  PROC DrawPart24()
    MoveL Offs(pOrigin,312.39,170.23,0.00),v60,z0,tPen\WObj:=wPaper;
    MoveL Offs(pOrigin,314.80,167.82,0.00),v40,z0,tPen\WObj:=wPaper;
    MoveL Offs(pOrigin,313.96,168.12,0.00),v40,z0,tPen\WObj:=wPaper;
    MoveL Offs(pOrigin,312.90,168.12,0.00),v40,fine,tPen\WObj:=wPaper;
    MoveL Offs(pOrigin,312.90,168.12,6.00),v60,z5,tPen\WObj:=wPaper;
    MoveL Offs(pOrigin,312.51,169.44,6.00),vTravel,z5,tPen\WObj:=wPaper;
    MoveL Offs(pOrigin,312.51,169.44,0.00),v60,z0,tPen\WObj:=wPaper;
    MoveL Offs(pOrigin,315.82,172.74,0.00),v40,z0,tPen\WObj:=wPaper;
    MoveL Offs(pOrigin,316.28,172.31,0.00),v40,z0,tPen\WObj:=wPaper;
    MoveL Offs(pOrigin,313.88,174.72,0.00),v40,z0,tPen\WObj:=wPaper;
    MoveL Offs(pOrigin,314.02,173.94,0.00),v40,z0,tPen\WObj:=wPaper;
    MoveL Offs(pOrigin,317.48,177.39,0.00),v40,z0,tPen\WObj:=wPaper;
    MoveL Offs(pOrigin,317.15,177.62,0.00),v40,z0,tPen\WObj:=wPaper;
    MoveL Offs(pOrigin,316.09,177.62,0.00),v40,z0,tPen\WObj:=wPaper;
    MoveL Offs(pOrigin,315.66,176.57,0.00),v40,z0,tPen\WObj:=wPaper;
    MoveL Offs(pOrigin,316.73,176.57,0.00),v40,z0,tPen\WObj:=wPaper;
    MoveL Offs(pOrigin,317.92,176.65,0.00),v40,z0,tPen\WObj:=wPaper;
    MoveL Offs(pOrigin,315.36,179.21,0.00),v40,z0,tPen\WObj:=wPaper;
    MoveL Offs(pOrigin,315.81,180.25,0.00),v40,z0,tPen\WObj:=wPaper;
    MoveL Offs(pOrigin,320.62,175.44,0.00),v40,z0,tPen\WObj:=wPaper;
    MoveL Offs(pOrigin,320.17,174.40,0.00),v40,z0,tPen\WObj:=wPaper;
    MoveL Offs(pOrigin,318.82,175.75,0.00),v40,fine,tPen\WObj:=wPaper;
    MoveL Offs(pOrigin,318.82,175.75,6.00),v60,z5,tPen\WObj:=wPaper;
    MoveL Offs(pOrigin,318.67,174.40,6.00),vTravel,z5,tPen\WObj:=wPaper;
    MoveL Offs(pOrigin,318.67,174.40,0.00),v60,z0,tPen\WObj:=wPaper;
    MoveL Offs(pOrigin,319.57,173.50,0.00),v40,fine,tPen\WObj:=wPaper;
    MoveL Offs(pOrigin,319.57,173.50,6.00),v60,z5,tPen\WObj:=wPaper;
    MoveL Offs(pOrigin,317.02,174.56,6.00),vTravel,z5,tPen\WObj:=wPaper;
    MoveL Offs(pOrigin,317.02,174.56,0.00),v60,z0,tPen\WObj:=wPaper;
    MoveL Offs(pOrigin,314.62,176.96,0.00),v40,z0,tPen\WObj:=wPaper;
    MoveL Offs(pOrigin,314.63,176.03,0.00),v40,z0,tPen\WObj:=wPaper;
    MoveL Offs(pOrigin,318.08,179.49,0.00),v40,z0,tPen\WObj:=wPaper;
    MoveL Offs(pOrigin,317.79,179.74,0.00),v40,z0,tPen\WObj:=wPaper;
    MoveL Offs(pOrigin,316.73,179.74,0.00),v40,z0,tPen\WObj:=wPaper;
    MoveL Offs(pOrigin,316.14,180.53,0.00),v40,z0,tPen\WObj:=wPaper;
    MoveL Offs(pOrigin,318.54,182.94,0.00),v40,z0,tPen\WObj:=wPaper;
    MoveL Offs(pOrigin,317.58,182.90,0.00),v40,z0,tPen\WObj:=wPaper;
    MoveL Offs(pOrigin,315.02,182.90,0.00),v40,z0,tPen\WObj:=wPaper;
    MoveL Offs(pOrigin,315.10,182.48,0.00),v40,z0,tPen\WObj:=wPaper;
    MoveL Offs(pOrigin,316.75,184.13,0.00),v40,fine,tPen\WObj:=wPaper;
    MoveL Offs(pOrigin,316.75,184.13,6.00),v60,z5,tPen\WObj:=wPaper;
    MoveL Offs(pOrigin,314.60,183.96,6.00),vTravel,z5,tPen\WObj:=wPaper;
    MoveL Offs(pOrigin,314.60,183.96,0.00),v60,z0,tPen\WObj:=wPaper;
    MoveL Offs(pOrigin,311.84,183.96,0.00),v40,z0,tPen\WObj:=wPaper;
    MoveL Offs(pOrigin,311.96,183.82,0.00),v40,z0,tPen\WObj:=wPaper;
    MoveL Offs(pOrigin,313.31,185.17,0.00),v40,z0,tPen\WObj:=wPaper;
    MoveL Offs(pOrigin,313.39,185.65,0.00),v40,z0,tPen\WObj:=wPaper;
    MoveL Offs(pOrigin,321.21,177.84,0.00),v40,fine,tPen\WObj:=wPaper;
    MoveL Offs(pOrigin,321.21,177.84,6.00),v60,z5,tPen\WObj:=wPaper;
    MoveL Offs(pOrigin,320.91,176.64,6.00),vTravel,z5,tPen\WObj:=wPaper;
    MoveL Offs(pOrigin,320.91,176.64,0.00),v60,z0,tPen\WObj:=wPaper;
    MoveL Offs(pOrigin,311.00,186.56,0.00),v40,z0,tPen\WObj:=wPaper;
    MoveL Offs(pOrigin,311.06,185.91,0.00),v40,z0,tPen\WObj:=wPaper;
    MoveL Offs(pOrigin,309.56,184.41,0.00),v40,z0,tPen\WObj:=wPaper;
    MoveL Offs(pOrigin,309.51,183.57,0.00),v40,z0,tPen\WObj:=wPaper;
    MoveL Offs(pOrigin,302.74,190.33,0.00),v40,z0,tPen\WObj:=wPaper;
    MoveL Offs(pOrigin,303.64,190.93,0.00),v40,z0,tPen\WObj:=wPaper;
    MoveL Offs(pOrigin,311.30,183.26,0.00),v40,z0,tPen\WObj:=wPaper;
    MoveL Offs(pOrigin,310.61,183.96,0.00),v40,z0,tPen\WObj:=wPaper;
    MoveL Offs(pOrigin,312.26,185.61,0.00),v40,z0,tPen\WObj:=wPaper;
    MoveL Offs(pOrigin,311.41,185.02,0.00),v40,z0,tPen\WObj:=wPaper;
    MoveL Offs(pOrigin,308.86,185.02,0.00),v40,z0,tPen\WObj:=wPaper;
    MoveL Offs(pOrigin,308.51,184.85,0.00),v40,z0,tPen\WObj:=wPaper;
    MoveL Offs(pOrigin,310.02,186.36,0.00),v40,fine,tPen\WObj:=wPaper;
    MoveL Offs(pOrigin,310.02,186.36,6.00),v60,z5,tPen\WObj:=wPaper;
    MoveL Offs(pOrigin,308.23,186.07,6.00),vTravel,z5,tPen\WObj:=wPaper;
    MoveL Offs(pOrigin,308.23,186.07,0.00),v60,z0,tPen\WObj:=wPaper;
    MoveL Offs(pOrigin,305.68,186.07,0.00),v40,z0,tPen\WObj:=wPaper;
    MoveL Offs(pOrigin,305.07,185.89,0.00),v40,z0,tPen\WObj:=wPaper;
    MoveL Offs(pOrigin,306.57,187.39,0.00),v40,z0,tPen\WObj:=wPaper;
    MoveL Offs(pOrigin,305.68,187.13,0.00),v40,z0,tPen\WObj:=wPaper;
    MoveL Offs(pOrigin,302.91,187.13,0.00),v40,z0,tPen\WObj:=wPaper;
    MoveL Offs(pOrigin,302.98,186.78,0.00),v40,z0,tPen\WObj:=wPaper;
    MoveL Offs(pOrigin,309.59,193.40,0.00),v40,z0,tPen\WObj:=wPaper;
    MoveL Offs(pOrigin,309.77,193.75,0.00),v40,z0,tPen\WObj:=wPaper;
    MoveL Offs(pOrigin,312.03,191.50,0.00),v40,z0,tPen\WObj:=wPaper;
    MoveL Offs(pOrigin,312.93,192.10,0.00),v40,z0,tPen\WObj:=wPaper;
    MoveL Offs(pOrigin,310.67,194.35,0.00),v40,z0,tPen\WObj:=wPaper;
    MoveL Offs(pOrigin,311.62,193.91,0.00),v40,z0,tPen\WObj:=wPaper;
    MoveL Offs(pOrigin,312.05,194.12,0.00),v40,z0,tPen\WObj:=wPaper;
    MoveL Offs(pOrigin,311.62,193.91,0.00),v40,z0,tPen\WObj:=wPaper;
    MoveL Offs(pOrigin,311.41,193.46,0.00),v40,z0,tPen\WObj:=wPaper;
    MoveL Offs(pOrigin,313.54,193.46,0.00),v40,z0,tPen\WObj:=wPaper;
    MoveL Offs(pOrigin,313.78,193.11,0.00),v40,z0,tPen\WObj:=wPaper;
    MoveL Offs(pOrigin,316.19,195.51,0.00),v40,z0,tPen\WObj:=wPaper;
    MoveL Offs(pOrigin,315.66,195.58,0.00),v40,z0,tPen\WObj:=wPaper;
    MoveL Offs(pOrigin,313.75,195.58,0.00),v40,z0,tPen\WObj:=wPaper;
    MoveL Offs(pOrigin,313.33,196.04,0.00),v40,z0,tPen\WObj:=wPaper;
    MoveL Offs(pOrigin,312.90,196.46,0.00),v40,z0,tPen\WObj:=wPaper;
    MoveL Offs(pOrigin,313.33,196.04,0.00),v40,z0,tPen\WObj:=wPaper;
    MoveL Offs(pOrigin,313.11,196.63,0.00),v40,z0,tPen\WObj:=wPaper;
    MoveL Offs(pOrigin,314.81,196.63,0.00),v40,z0,tPen\WObj:=wPaper;
    MoveL Offs(pOrigin,314.84,197.16,0.00),v40,z0,tPen\WObj:=wPaper;
    MoveL Offs(pOrigin,307.78,190.09,0.00),v40,z0,tPen\WObj:=wPaper;
    MoveL Offs(pOrigin,307.99,189.56,0.00),v40,z0,tPen\WObj:=wPaper;
    MoveL Offs(pOrigin,305.59,191.97,0.00),v40,z0,tPen\WObj:=wPaper;
    MoveL Offs(pOrigin,306.59,191.89,0.00),v40,z0,tPen\WObj:=wPaper;
    MoveL Offs(pOrigin,301.93,187.23,0.00),v40,z0,tPen\WObj:=wPaper;
    MoveL Offs(pOrigin,302.31,186.29,0.00),v40,z0,tPen\WObj:=wPaper;
    MoveL Offs(pOrigin,289.84,198.76,0.00),v40,z0,tPen\WObj:=wPaper;
    MoveL Offs(pOrigin,289.23,198.43,0.00),v40,z0,tPen\WObj:=wPaper;
    MoveL Offs(pOrigin,288.48,197.68,0.00),v40,z0,tPen\WObj:=wPaper;
    MoveL Offs(pOrigin,289.23,196.93,0.00),v40,z0,tPen\WObj:=wPaper;
    MoveL Offs(pOrigin,290.28,197.98,0.00),v40,z0,tPen\WObj:=wPaper;
    MoveL Offs(pOrigin,291.03,197.23,0.00),v40,z0,tPen\WObj:=wPaper;
    MoveL Offs(pOrigin,290.12,196.33,0.00),v40,z0,tPen\WObj:=wPaper;
    MoveL Offs(pOrigin,290.87,195.59,0.00),v40,z0,tPen\WObj:=wPaper;
    MoveL Offs(pOrigin,291.92,196.64,0.00),v40,z0,tPen\WObj:=wPaper;
    MoveL Offs(pOrigin,292.67,195.89,0.00),v40,z0,tPen\WObj:=wPaper;
    MoveL Offs(pOrigin,291.77,194.99,0.00),v40,z0,tPen\WObj:=wPaper;
    MoveL Offs(pOrigin,292.51,194.24,0.00),v40,z0,tPen\WObj:=wPaper;
    MoveL Offs(pOrigin,293.57,195.29,0.00),v40,z0,tPen\WObj:=wPaper;
    MoveL Offs(pOrigin,293.35,194.34,0.00),v40,z0,tPen\WObj:=wPaper;
    MoveL Offs(pOrigin,287.40,199.23,0.00),v40,z0,tPen\WObj:=wPaper;
    MoveL Offs(pOrigin,289.74,212.19,0.00),v40,z0,tPen\WObj:=wPaper;
    MoveL Offs(pOrigin,289.95,218.14,0.00),v40,z0,tPen\WObj:=wPaper;
    MoveL Offs(pOrigin,289.52,223.24,0.00),v40,z0,tPen\WObj:=wPaper;
    MoveL Offs(pOrigin,289.52,223.24,0.00),v40,z0,tPen\WObj:=wPaper;
    MoveL Offs(pOrigin,290.80,222.60,0.00),v40,z0,tPen\WObj:=wPaper;
    MoveL Offs(pOrigin,294.20,218.35,0.00),v40,z0,tPen\WObj:=wPaper;
  ENDPROC

  PROC DrawPart25()
    MoveL Offs(pOrigin,301.21,211.34,0.00),v40,z0,tPen\WObj:=wPaper;
    MoveL Offs(pOrigin,313.75,195.61,0.00),v40,z0,tPen\WObj:=wPaper;
    MoveL Offs(pOrigin,313.68,194.76,0.00),v40,z0,tPen\WObj:=wPaper;
    MoveL Offs(pOrigin,302.06,189.24,0.00),v40,z0,tPen\WObj:=wPaper;
    MoveL Offs(pOrigin,300.79,189.38,0.00),v40,z0,tPen\WObj:=wPaper;
    MoveL Offs(pOrigin,297.81,191.22,0.00),v40,z0,tPen\WObj:=wPaper;
    MoveL Offs(pOrigin,297.32,190.94,0.00),v40,z0,tPen\WObj:=wPaper;
    MoveL Offs(pOrigin,297.39,190.51,0.00),v40,z0,tPen\WObj:=wPaper;
    MoveL Offs(pOrigin,302.27,187.47,0.00),v40,z0,tPen\WObj:=wPaper;
    MoveL Offs(pOrigin,316.94,182.23,0.00),v40,z0,tPen\WObj:=wPaper;
    MoveL Offs(pOrigin,317.15,181.59,0.00),v40,z0,tPen\WObj:=wPaper;
    MoveL Offs(pOrigin,309.71,159.27,0.00),v40,z0,tPen\WObj:=wPaper;
    MoveL Offs(pOrigin,291.65,101.26,0.00),v40,z0,tPen\WObj:=wPaper;
    MoveL Offs(pOrigin,286.98,81.71,0.00),v40,z0,tPen\WObj:=wPaper;
    MoveL Offs(pOrigin,285.49,73.21,0.00),v40,z0,tPen\WObj:=wPaper;
    MoveL Offs(pOrigin,285.06,68.75,0.00),v40,z0,tPen\WObj:=wPaper;
    MoveL Offs(pOrigin,281.88,68.54,0.00),v40,z0,tPen\WObj:=wPaper;
    MoveL Offs(pOrigin,276.14,66.62,0.00),v40,z0,tPen\WObj:=wPaper;
    MoveL Offs(pOrigin,275.50,68.54,0.00),v40,z0,tPen\WObj:=wPaper;
    MoveL Offs(pOrigin,273.59,80.44,0.00),v40,z0,tPen\WObj:=wPaper;
    MoveL Offs(pOrigin,272.31,92.97,0.00),v40,z0,tPen\WObj:=wPaper;
    MoveL Offs(pOrigin,271.89,100.41,0.00),v40,z0,tPen\WObj:=wPaper;
    MoveL Offs(pOrigin,271.89,111.68,0.00),v40,z0,tPen\WObj:=wPaper;
    MoveL Offs(pOrigin,272.52,122.30,0.00),v40,z0,tPen\WObj:=wPaper;
    MoveL Offs(pOrigin,274.23,137.18,0.00),v40,z0,tPen\WObj:=wPaper;
    MoveL Offs(pOrigin,277.62,157.57,0.00),v40,z0,tPen\WObj:=wPaper;
    MoveL Offs(pOrigin,281.45,175.64,0.00),v40,z0,tPen\WObj:=wPaper;
    MoveL Offs(pOrigin,286.98,197.74,0.00),v40,z0,tPen\WObj:=wPaper;
    MoveL Offs(pOrigin,287.61,198.59,0.00),v40,z0,tPen\WObj:=wPaper;
    MoveL Offs(pOrigin,287.61,198.74,0.00),v40,z0,tPen\WObj:=wPaper;
    MoveL Offs(pOrigin,285.91,198.74,0.00),v40,z0,tPen\WObj:=wPaper;
    MoveL Offs(pOrigin,285.34,199.01,0.00),v40,z0,tPen\WObj:=wPaper;
    MoveL Offs(pOrigin,288.34,202.02,0.00),v40,z0,tPen\WObj:=wPaper;
    MoveL Offs(pOrigin,287.82,201.91,0.00),v40,z0,tPen\WObj:=wPaper;
    MoveL Offs(pOrigin,286.76,201.91,0.00),v40,z0,tPen\WObj:=wPaper;
    MoveL Offs(pOrigin,286.98,202.97,0.00),v40,z0,tPen\WObj:=wPaper;
    MoveL Offs(pOrigin,288.04,202.97,0.00),v40,z0,tPen\WObj:=wPaper;
    MoveL Offs(pOrigin,288.93,202.66,0.00),v40,z0,tPen\WObj:=wPaper;
    MoveL Offs(pOrigin,286.37,205.21,0.00),v40,z0,tPen\WObj:=wPaper;
    MoveL Offs(pOrigin,286.55,204.71,0.00),v40,z0,tPen\WObj:=wPaper;
    MoveL Offs(pOrigin,289.26,207.41,0.00),v40,z0,tPen\WObj:=wPaper;
    MoveL Offs(pOrigin,288.89,207.19,0.00),v40,z0,tPen\WObj:=wPaper;
    MoveL Offs(pOrigin,287.82,207.19,0.00),v40,z0,tPen\WObj:=wPaper;
    MoveL Offs(pOrigin,287.61,206.14,0.00),v40,z0,tPen\WObj:=wPaper;
    MoveL Offs(pOrigin,288.68,206.14,0.00),v40,z0,tPen\WObj:=wPaper;
    MoveL Offs(pOrigin,288.95,205.62,0.00),v40,z0,tPen\WObj:=wPaper;
    MoveL Offs(pOrigin,286.25,202.91,0.00),v40,z0,tPen\WObj:=wPaper;
    MoveL Offs(pOrigin,285.78,202.82,0.00),v40,z0,tPen\WObj:=wPaper;
    MoveL Offs(pOrigin,288.63,199.96,0.00),v40,z0,tPen\WObj:=wPaper;
    MoveL Offs(pOrigin,287.89,200.07,0.00),v40,z0,tPen\WObj:=wPaper;
    MoveL Offs(pOrigin,284.73,196.92,0.00),v40,z0,tPen\WObj:=wPaper;
    MoveL Offs(pOrigin,284.30,196.83,0.00),v40,z0,tPen\WObj:=wPaper;
    MoveL Offs(pOrigin,287.00,194.12,0.00),v40,z0,tPen\WObj:=wPaper;
    MoveL Offs(pOrigin,286.37,194.07,0.00),v40,z0,tPen\WObj:=wPaper;
    MoveL Offs(pOrigin,283.22,190.92,0.00),v40,z0,tPen\WObj:=wPaper;
    MoveL Offs(pOrigin,282.82,190.84,0.00),v40,z0,tPen\WObj:=wPaper;
    MoveL Offs(pOrigin,285.37,188.29,0.00),v40,z0,tPen\WObj:=wPaper;
    MoveL Offs(pOrigin,285.16,188.38,0.00),v40,z0,tPen\WObj:=wPaper;
    MoveL Offs(pOrigin,281.85,185.07,0.00),v40,z0,tPen\WObj:=wPaper;
    MoveL Offs(pOrigin,281.34,184.85,0.00),v40,z0,tPen\WObj:=wPaper;
    MoveL Offs(pOrigin,283.89,182.30,0.00),v40,z0,tPen\WObj:=wPaper;
    MoveL Offs(pOrigin,283.64,182.38,0.00),v40,z0,tPen\WObj:=wPaper;
    MoveL Offs(pOrigin,277.93,176.67,0.00),v40,z0,tPen\WObj:=wPaper;
    MoveL Offs(pOrigin,278.90,176.57,0.00),v40,z0,tPen\WObj:=wPaper;
    MoveL Offs(pOrigin,281.66,176.57,0.00),v40,z0,tPen\WObj:=wPaper;
    MoveL Offs(pOrigin,282.12,176.38,0.00),v40,z0,tPen\WObj:=wPaper;
    MoveL Offs(pOrigin,279.12,173.38,0.00),v40,z0,tPen\WObj:=wPaper;
    MoveL Offs(pOrigin,279.75,173.40,0.00),v40,z0,tPen\WObj:=wPaper;
    MoveL Offs(pOrigin,280.81,173.40,0.00),v40,z0,tPen\WObj:=wPaper;
    MoveL Offs(pOrigin,281.21,172.49,0.00),v40,z0,tPen\WObj:=wPaper;
    MoveL Offs(pOrigin,278.21,169.48,0.00),v40,z0,tPen\WObj:=wPaper;
    MoveL Offs(pOrigin,277.64,169.14,0.00),v40,z0,tPen\WObj:=wPaper;
    MoveL Offs(pOrigin,280.35,166.43,0.00),v40,z0,tPen\WObj:=wPaper;
    MoveL Offs(pOrigin,280.00,166.79,0.00),v40,z0,tPen\WObj:=wPaper;
    MoveL Offs(pOrigin,276.84,163.64,0.00),v40,z0,tPen\WObj:=wPaper;
    MoveL Offs(pOrigin,276.61,164.20,0.00),v40,z0,tPen\WObj:=wPaper;
    MoveL Offs(pOrigin,279.16,161.64,0.00),v40,z0,tPen\WObj:=wPaper;
    MoveL Offs(pOrigin,278.93,161.25,0.00),v40,z0,tPen\WObj:=wPaper;
    MoveL Offs(pOrigin,275.78,158.09,0.00),v40,z0,tPen\WObj:=wPaper;
    MoveL Offs(pOrigin,275.28,158.06,0.00),v40,z0,tPen\WObj:=wPaper;
    MoveL Offs(pOrigin,278.14,155.20,0.00),v40,z0,tPen\WObj:=wPaper;
    MoveL Offs(pOrigin,277.72,155.55,0.00),v40,z0,tPen\WObj:=wPaper;
    MoveL Offs(pOrigin,273.66,151.49,0.00),v40,z0,tPen\WObj:=wPaper;
    MoveL Offs(pOrigin,273.05,151.32,0.00),v40,z0,tPen\WObj:=wPaper;
    MoveL Offs(pOrigin,276.96,147.42,0.00),v40,z0,tPen\WObj:=wPaper;
    MoveL Offs(pOrigin,276.49,148.35,0.00),v40,z0,tPen\WObj:=wPaper;
    MoveL Offs(pOrigin,273.49,145.35,0.00),v40,z0,tPen\WObj:=wPaper;
    MoveL Offs(pOrigin,274.44,145.94,0.00),v40,z0,tPen\WObj:=wPaper;
    MoveL Offs(pOrigin,275.50,145.94,0.00),v40,z0,tPen\WObj:=wPaper;
    MoveL Offs(pOrigin,276.04,146.41,0.00),v40,z0,tPen\WObj:=wPaper;
    MoveL Offs(pOrigin,273.18,143.55,0.00),v40,z0,tPen\WObj:=wPaper;
    MoveL Offs(pOrigin,274.01,142.78,0.00),v40,z0,tPen\WObj:=wPaper;
    MoveL Offs(pOrigin,275.08,142.78,0.00),v40,z0,tPen\WObj:=wPaper;
    MoveL Offs(pOrigin,275.58,142.96,0.00),v40,z0,tPen\WObj:=wPaper;
    MoveL Offs(pOrigin,272.87,140.25,0.00),v40,z0,tPen\WObj:=wPaper;
    MoveL Offs(pOrigin,272.34,140.09,0.00),v40,z0,tPen\WObj:=wPaper;
    MoveL Offs(pOrigin,275.19,137.24,0.00),v40,z0,tPen\WObj:=wPaper;
    MoveL Offs(pOrigin,274.81,137.71,0.00),v40,z0,tPen\WObj:=wPaper;
    MoveL Offs(pOrigin,271.96,134.86,0.00),v40,z0,tPen\WObj:=wPaper;
    MoveL Offs(pOrigin,271.61,134.85,0.00),v40,z0,tPen\WObj:=wPaper;
    MoveL Offs(pOrigin,274.46,131.99,0.00),v40,z0,tPen\WObj:=wPaper;
    MoveL Offs(pOrigin,273.90,132.32,0.00),v40,z0,tPen\WObj:=wPaper;
    MoveL Offs(pOrigin,271.34,129.76,0.00),v40,z0,tPen\WObj:=wPaper;
    MoveL Offs(pOrigin,271.02,129.46,0.00),v40,z0,tPen\WObj:=wPaper;
    MoveL Offs(pOrigin,274.03,126.45,0.00),v40,z0,tPen\WObj:=wPaper;
    MoveL Offs(pOrigin,273.43,125.88,0.00),v40,z0,tPen\WObj:=wPaper;
    MoveL Offs(pOrigin,270.73,123.17,0.00),v40,z0,tPen\WObj:=wPaper;
    MoveL Offs(pOrigin,270.30,122.72,0.00),v40,z0,tPen\WObj:=wPaper;
    MoveL Offs(pOrigin,273.30,119.71,0.00),v40,z0,tPen\WObj:=wPaper;
    MoveL Offs(pOrigin,272.81,119.28,0.00),v40,z0,tPen\WObj:=wPaper;
    MoveL Offs(pOrigin,270.11,116.58,0.00),v40,z0,tPen\WObj:=wPaper;
    MoveL Offs(pOrigin,269.56,117.48,0.00),v40,z0,tPen\WObj:=wPaper;
    MoveL Offs(pOrigin,272.87,114.17,0.00),v40,z0,tPen\WObj:=wPaper;
    MoveL Offs(pOrigin,272.50,114.49,0.00),v40,z0,tPen\WObj:=wPaper;
    MoveL Offs(pOrigin,270.09,112.08,0.00),v40,z0,tPen\WObj:=wPaper;
    MoveL Offs(pOrigin,269.43,111.64,0.00),v40,z0,tPen\WObj:=wPaper;
    MoveL Offs(pOrigin,272.74,108.33,0.00),v40,z0,tPen\WObj:=wPaper;
    MoveL Offs(pOrigin,272.33,108.35,0.00),v40,z0,tPen\WObj:=wPaper;
    MoveL Offs(pOrigin,269.92,105.94,0.00),v40,z0,tPen\WObj:=wPaper;
    MoveL Offs(pOrigin,269.45,105.65,0.00),v40,z0,tPen\WObj:=wPaper;
  ENDPROC

  PROC DrawPart26()
    MoveL Offs(pOrigin,272.76,102.34,0.00),v40,z0,tPen\WObj:=wPaper;
    MoveL Offs(pOrigin,272.31,102.35,0.00),v40,z0,tPen\WObj:=wPaper;
    MoveL Offs(pOrigin,270.06,100.10,0.00),v40,z0,tPen\WObj:=wPaper;
    MoveL Offs(pOrigin,270.61,100.54,0.00),v40,z0,tPen\WObj:=wPaper;
    MoveL Offs(pOrigin,271.68,100.54,0.00),v40,z0,tPen\WObj:=wPaper;
    MoveL Offs(pOrigin,272.30,100.86,0.00),v40,z0,tPen\WObj:=wPaper;
    MoveL Offs(pOrigin,270.05,98.60,0.00),v40,z0,tPen\WObj:=wPaper;
    MoveL Offs(pOrigin,269.62,98.01,0.00),v40,z0,tPen\WObj:=wPaper;
    MoveL Offs(pOrigin,273.08,94.55,0.00),v40,z0,tPen\WObj:=wPaper;
    MoveL Offs(pOrigin,272.44,95.01,0.00),v40,z0,tPen\WObj:=wPaper;
    MoveL Offs(pOrigin,270.33,92.91,0.00),v40,z0,tPen\WObj:=wPaper;
    MoveL Offs(pOrigin,269.94,93.21,0.00),v40,z0,tPen\WObj:=wPaper;
    MoveL Offs(pOrigin,273.54,89.60,0.00),v40,z0,tPen\WObj:=wPaper;
    MoveL Offs(pOrigin,273.02,89.62,0.00),v40,z0,tPen\WObj:=wPaper;
    MoveL Offs(pOrigin,270.92,87.52,0.00),v40,z0,tPen\WObj:=wPaper;
    MoveL Offs(pOrigin,271.46,87.86,0.00),v40,z0,tPen\WObj:=wPaper;
    MoveL Offs(pOrigin,272.74,87.86,0.00),v40,z0,tPen\WObj:=wPaper;
    MoveL Offs(pOrigin,272.74,86.81,0.00),v40,z0,tPen\WObj:=wPaper;
    MoveL Offs(pOrigin,271.68,86.81,0.00),v40,z0,tPen\WObj:=wPaper;
    MoveL Offs(pOrigin,271.68,85.75,0.00),v40,z0,tPen\WObj:=wPaper;
    MoveL Offs(pOrigin,272.95,85.75,0.00),v40,z0,tPen\WObj:=wPaper;
    MoveL Offs(pOrigin,273.31,85.43,0.00),v40,z0,tPen\WObj:=wPaper;
    MoveL Offs(pOrigin,271.35,83.48,0.00),v40,z0,tPen\WObj:=wPaper;
    MoveL Offs(pOrigin,271.89,83.64,0.00),v40,z0,tPen\WObj:=wPaper;
    MoveL Offs(pOrigin,273.16,83.64,0.00),v40,z0,tPen\WObj:=wPaper;
    MoveL Offs(pOrigin,273.45,84.08,0.00),v40,z0,tPen\WObj:=wPaper;
    MoveL Offs(pOrigin,271.35,81.98,0.00),v40,z0,tPen\WObj:=wPaper;
    MoveL Offs(pOrigin,270.72,81.97,0.00),v40,z0,tPen\WObj:=wPaper;
    MoveL Offs(pOrigin,275.08,77.62,0.00),v40,fine,tPen\WObj:=wPaper;
    MoveL Offs(pOrigin,275.08,77.62,6.00),v60,z5,tPen\WObj:=wPaper;
    MoveL Offs(pOrigin,274.01,76.25,6.00),vTravel,z5,tPen\WObj:=wPaper;
    MoveL Offs(pOrigin,274.01,76.25,0.00),v60,z0,tPen\WObj:=wPaper;
    MoveL Offs(pOrigin,272.95,76.25,0.00),v40,z0,tPen\WObj:=wPaper;
    MoveL Offs(pOrigin,272.95,75.19,0.00),v40,z0,tPen\WObj:=wPaper;
    MoveL Offs(pOrigin,274.23,75.19,0.00),v40,z0,tPen\WObj:=wPaper;
    MoveL Offs(pOrigin,274.92,75.10,0.00),v40,z0,tPen\WObj:=wPaper;
    MoveL Offs(pOrigin,272.82,72.99,0.00),v40,z0,tPen\WObj:=wPaper;
    MoveL Offs(pOrigin,272.10,73.13,0.00),v40,z0,tPen\WObj:=wPaper;
    MoveL Offs(pOrigin,276.30,68.92,0.00),v40,z0,tPen\WObj:=wPaper;
    MoveL Offs(pOrigin,275.95,68.66,0.00),v40,z0,tPen\WObj:=wPaper;
    MoveL Offs(pOrigin,273.70,66.41,0.00),v40,z0,tPen\WObj:=wPaper;
    MoveL Offs(pOrigin,273.02,66.24,0.00),v40,z0,tPen\WObj:=wPaper;
    MoveL Offs(pOrigin,275.57,63.68,0.00),v40,z0,tPen\WObj:=wPaper;
    MoveL Offs(pOrigin,275.71,64.63,0.00),v40,z0,tPen\WObj:=wPaper;
    MoveL Offs(pOrigin,272.74,64.63,0.00),v40,z0,tPen\WObj:=wPaper;
    MoveL Offs(pOrigin,272.65,65.35,0.00),v40,z0,tPen\WObj:=wPaper;
    MoveL Offs(pOrigin,266.94,59.64,0.00),v40,z0,tPen\WObj:=wPaper;
    MoveL Offs(pOrigin,267.85,59.35,0.00),v40,z0,tPen\WObj:=wPaper;
    MoveL Offs(pOrigin,269.12,59.35,0.00),v40,fine,tPen\WObj:=wPaper;
    MoveL Offs(pOrigin,269.12,59.35,6.00),v60,z5,tPen\WObj:=wPaper;
    MoveL Offs(pOrigin,267.53,58.75,6.00),vTravel,z5,tPen\WObj:=wPaper;
    MoveL Offs(pOrigin,267.53,58.75,0.00),v60,z0,tPen\WObj:=wPaper;
    MoveL Offs(pOrigin,276.40,67.61,0.00),v40,z0,tPen\WObj:=wPaper;
    MoveL Offs(pOrigin,277.20,68.02,0.00),v40,z0,tPen\WObj:=wPaper;
    MoveL Offs(pOrigin,279.91,65.32,0.00),v40,z0,tPen\WObj:=wPaper;
    MoveL Offs(pOrigin,280.96,65.76,0.00),v40,z0,tPen\WObj:=wPaper;
    MoveL Offs(pOrigin,278.55,68.17,0.00),v40,z0,tPen\WObj:=wPaper;
    MoveL Offs(pOrigin,278.05,67.77,0.00),v40,z0,tPen\WObj:=wPaper;
    MoveL Offs(pOrigin,273.54,63.26,0.00),v40,z0,tPen\WObj:=wPaper;
    MoveL Offs(pOrigin,273.16,63.58,0.00),v40,z0,tPen\WObj:=wPaper;
    MoveL Offs(pOrigin,270.40,63.58,0.00),v40,z0,tPen\WObj:=wPaper;
    MoveL Offs(pOrigin,270.35,63.22,0.00),v40,z0,tPen\WObj:=wPaper;
    MoveL Offs(pOrigin,270.35,61.74,0.00),v40,fine,tPen\WObj:=wPaper;
    MoveL Offs(pOrigin,270.35,61.74,6.00),v60,z5,tPen\WObj:=wPaper;
    MoveL Offs(pOrigin,271.68,62.52,6.00),vTravel,z5,tPen\WObj:=wPaper;
    MoveL Offs(pOrigin,271.68,62.52,0.00),v60,z0,tPen\WObj:=wPaper;
    MoveL Offs(pOrigin,267.64,62.52,0.00),v40,z0,tPen\WObj:=wPaper;
    MoveL Offs(pOrigin,267.55,63.24,0.00),v40,z0,tPen\WObj:=wPaper;
    MoveL Offs(pOrigin,262.59,58.28,0.00),v40,z0,tPen\WObj:=wPaper;
    MoveL Offs(pOrigin,263.15,58.18,0.00),v40,z0,tPen\WObj:=wPaper;
    MoveL Offs(pOrigin,260.90,60.43,0.00),v40,z0,tPen\WObj:=wPaper;
    MoveL Offs(pOrigin,261.80,61.03,0.00),v40,z0,tPen\WObj:=wPaper;
    MoveL Offs(pOrigin,264.20,58.62,0.00),v40,fine,tPen\WObj:=wPaper;
    MoveL Offs(pOrigin,264.20,58.62,6.00),v60,z5,tPen\WObj:=wPaper;
    MoveL Offs(pOrigin,263.18,59.35,6.00),vTravel,z5,tPen\WObj:=wPaper;
    MoveL Offs(pOrigin,263.18,59.35,0.00),v60,z0,tPen\WObj:=wPaper;
    MoveL Offs(pOrigin,260.84,59.35,0.00),v40,z0,tPen\WObj:=wPaper;
    MoveL Offs(pOrigin,261.26,58.34,0.00),v40,z0,tPen\WObj:=wPaper;
    MoveL Offs(pOrigin,261.69,58.55,0.00),v40,z0,tPen\WObj:=wPaper;
    MoveL Offs(pOrigin,261.26,58.34,0.00),v40,z0,tPen\WObj:=wPaper;
    MoveL Offs(pOrigin,261.26,58.30,0.00),v40,z0,tPen\WObj:=wPaper;
    MoveL Offs(pOrigin,259.35,58.30,0.00),v40,z0,tPen\WObj:=wPaper;
    MoveL Offs(pOrigin,259.56,57.24,0.00),v40,z0,tPen\WObj:=wPaper;
    MoveL Offs(pOrigin,257.86,57.24,0.00),v40,z0,tPen\WObj:=wPaper;
    MoveL Offs(pOrigin,257.31,58.05,0.00),v40,z0,tPen\WObj:=wPaper;
    MoveL Offs(pOrigin,259.57,55.79,0.00),v40,z0,tPen\WObj:=wPaper;
    MoveL Offs(pOrigin,258.82,55.05,0.00),v40,z0,tPen\WObj:=wPaper;
    MoveL Offs(pOrigin,256.41,57.45,0.00),v40,fine,tPen\WObj:=wPaper;
    MoveL Offs(pOrigin,256.41,57.45,6.00),v60,z5,tPen\WObj:=wPaper;
    MoveL Offs(pOrigin,256.59,56.18,6.00),vTravel,z5,tPen\WObj:=wPaper;
    MoveL Offs(pOrigin,256.59,56.18,0.00),v60,z0,tPen\WObj:=wPaper;
    MoveL Offs(pOrigin,258.29,56.18,0.00),v40,fine,tPen\WObj:=wPaper;
    MoveL Offs(pOrigin,258.29,56.18,6.00),v60,z5,tPen\WObj:=wPaper;
    MoveL Offs(pOrigin,257.92,54.45,6.00),vTravel,z5,tPen\WObj:=wPaper;
    MoveL Offs(pOrigin,257.92,54.45,0.00),v60,z0,tPen\WObj:=wPaper;
    MoveL Offs(pOrigin,254.92,57.45,0.00),v40,fine,tPen\WObj:=wPaper;
    MoveL Offs(pOrigin,254.92,57.45,6.00),v60,z5,tPen\WObj:=wPaper;
    MoveL Offs(pOrigin,254.62,56.26,6.00),vTravel,z5,tPen\WObj:=wPaper;
    MoveL Offs(pOrigin,254.62,56.26,0.00),v60,z0,tPen\WObj:=wPaper;
    MoveL Offs(pOrigin,257.03,53.85,0.00),v40,z0,tPen\WObj:=wPaper;
    MoveL Offs(pOrigin,255.95,53.88,0.00),v40,z0,tPen\WObj:=wPaper;
    MoveL Offs(pOrigin,256.38,54.30,0.00),v40,z0,tPen\WObj:=wPaper;
    MoveL Offs(pOrigin,255.95,53.88,0.00),v40,z0,tPen\WObj:=wPaper;
    MoveL Offs(pOrigin,255.95,54.07,0.00),v40,z0,tPen\WObj:=wPaper;
    MoveL Offs(pOrigin,254.25,54.07,0.00),v40,z0,tPen\WObj:=wPaper;
    MoveL Offs(pOrigin,253.28,54.61,0.00),v40,z0,tPen\WObj:=wPaper;
    MoveL Offs(pOrigin,255.53,52.36,0.00),v40,z0,tPen\WObj:=wPaper;
    MoveL Offs(pOrigin,254.89,53.02,0.00),v40,z0,tPen\WObj:=wPaper;
    MoveL Offs(pOrigin,253.19,53.02,0.00),v40,z0,tPen\WObj:=wPaper;
    MoveL Offs(pOrigin,252.53,53.87,0.00),v40,z0,tPen\WObj:=wPaper;
    MoveL Offs(pOrigin,254.94,51.46,0.00),v40,z0,tPen\WObj:=wPaper;
    MoveL Offs(pOrigin,254.04,50.87,0.00),v40,z0,tPen\WObj:=wPaper;
    MoveL Offs(pOrigin,251.93,52.97,0.00),v40,z0,tPen\WObj:=wPaper;
    MoveL Offs(pOrigin,252.12,51.96,0.00),v40,z0,tPen\WObj:=wPaper;
    MoveL Offs(pOrigin,253.82,51.96,0.00),v40,z0,tPen\WObj:=wPaper;
    MoveL Offs(pOrigin,253.40,51.54,0.00),v40,z0,tPen\WObj:=wPaper;
    MoveL Offs(pOrigin,255.10,53.24,0.00),v40,z0,tPen\WObj:=wPaper;
    MoveL Offs(pOrigin,253.40,51.54,0.00),v40,z0,tPen\WObj:=wPaper;
    MoveL Offs(pOrigin,252.98,50.90,0.00),v40,z0,tPen\WObj:=wPaper;
    MoveL Offs(pOrigin,251.28,50.90,0.00),v40,z0,tPen\WObj:=wPaper;
  ENDPROC

  PROC DrawPart27()
    MoveL Offs(pOrigin,250.44,51.48,0.00),v40,z0,tPen\WObj:=wPaper;
    MoveL Offs(pOrigin,252.54,49.37,0.00),v40,z0,tPen\WObj:=wPaper;
    MoveL Offs(pOrigin,251.91,49.85,0.00),v40,z0,tPen\WObj:=wPaper;
    MoveL Offs(pOrigin,250.42,49.85,0.00),v40,z0,tPen\WObj:=wPaper;
    MoveL Offs(pOrigin,250.00,50.05,0.00),v40,z0,tPen\WObj:=wPaper;
    MoveL Offs(pOrigin,254.25,54.30,0.00),v40,z0,tPen\WObj:=wPaper;
    MoveL Offs(pOrigin,250.00,50.05,0.00),v40,z0,tPen\WObj:=wPaper;
    MoveL Offs(pOrigin,249.69,50.73,0.00),v40,z0,tPen\WObj:=wPaper;
    MoveL Offs(pOrigin,251.95,48.48,0.00),v40,z0,tPen\WObj:=wPaper;
    MoveL Offs(pOrigin,251.05,47.88,0.00),v40,z0,tPen\WObj:=wPaper;
    MoveL Offs(pOrigin,248.95,49.98,0.00),v40,z0,tPen\WObj:=wPaper;
    MoveL Offs(pOrigin,248.20,49.24,0.00),v40,z0,tPen\WObj:=wPaper;
    MoveL Offs(pOrigin,250.46,46.98,0.00),v40,z0,tPen\WObj:=wPaper;
    MoveL Offs(pOrigin,250.27,47.46,0.00),v40,z0,tPen\WObj:=wPaper;
    MoveL Offs(pOrigin,240.80,37.99,0.00),v40,z0,tPen\WObj:=wPaper;
    MoveL Offs(pOrigin,241.29,38.23,0.00),v40,z0,tPen\WObj:=wPaper;
    MoveL Offs(pOrigin,242.78,38.23,0.00),v40,z0,tPen\WObj:=wPaper;
    MoveL Offs(pOrigin,243.20,37.40,0.00),v40,z0,tPen\WObj:=wPaper;
    MoveL Offs(pOrigin,241.40,35.60,0.00),v40,z0,tPen\WObj:=wPaper;
    MoveL Offs(pOrigin,241.93,35.60,0.00),v40,z0,tPen\WObj:=wPaper;
    MoveL Offs(pOrigin,242.14,35.17,0.00),v40,z0,tPen\WObj:=wPaper;
    MoveL Offs(pOrigin,241.93,35.60,0.00),v40,z0,tPen\WObj:=wPaper;
    MoveL Offs(pOrigin,241.71,36.12,0.00),v40,z0,tPen\WObj:=wPaper;
    MoveL Offs(pOrigin,243.41,36.12,0.00),v40,z0,tPen\WObj:=wPaper;
    MoveL Offs(pOrigin,243.41,35.60,0.00),v40,z0,tPen\WObj:=wPaper;
    MoveL Offs(pOrigin,242.99,36.24,0.00),v40,z0,tPen\WObj:=wPaper;
    MoveL Offs(pOrigin,243.41,35.60,0.00),v40,z0,tPen\WObj:=wPaper;
    MoveL Offs(pOrigin,243.95,35.39,0.00),v40,z0,tPen\WObj:=wPaper;
    MoveL Offs(pOrigin,243.95,34.11,0.00),v40,fine,tPen\WObj:=wPaper;
    MoveL Offs(pOrigin,243.95,34.11,6.00),v60,z5,tPen\WObj:=wPaper;
    MoveL Offs(pOrigin,245.96,31.99,6.00),vTravel,z5,tPen\WObj:=wPaper;
    MoveL Offs(pOrigin,245.96,31.99,0.00),v60,z0,tPen\WObj:=wPaper;
    MoveL Offs(pOrigin,245.75,32.41,0.00),v40,z0,tPen\WObj:=wPaper;
    MoveL Offs(pOrigin,245.96,31.99,0.00),v40,z0,tPen\WObj:=wPaper;
    MoveL Offs(pOrigin,245.11,31.35,0.00),v40,z0,tPen\WObj:=wPaper;
    MoveL Offs(pOrigin,245.32,30.92,0.00),v40,z0,tPen\WObj:=wPaper;
    MoveL Offs(pOrigin,245.11,31.35,0.00),v40,fine,tPen\WObj:=wPaper;
    MoveL Offs(pOrigin,245.11,31.35,6.00),v60,z5,tPen\WObj:=wPaper;
    MoveL Offs(pOrigin,246.02,29.77,6.00),vTravel,z5,tPen\WObj:=wPaper;
    MoveL Offs(pOrigin,246.02,29.77,0.00),v60,z0,tPen\WObj:=wPaper;
    MoveL Offs(pOrigin,247.97,31.72,0.00),v40,z0,tPen\WObj:=wPaper;
    MoveL Offs(pOrigin,248.85,32.16,0.00),v40,z0,tPen\WObj:=wPaper;
    MoveL Offs(pOrigin,252.61,28.40,0.00),v40,fine,tPen\WObj:=wPaper;
    MoveL Offs(pOrigin,252.61,28.40,6.00),v60,z5,tPen\WObj:=wPaper;
    MoveL Offs(pOrigin,254.26,28.25,6.00),vTravel,z5,tPen\WObj:=wPaper;
    MoveL Offs(pOrigin,254.26,28.25,0.00),v60,z0,tPen\WObj:=wPaper;
    MoveL Offs(pOrigin,249.90,32.60,0.00),v40,z0,tPen\WObj:=wPaper;
    MoveL Offs(pOrigin,250.80,33.20,0.00),v40,z0,tPen\WObj:=wPaper;
    MoveL Offs(pOrigin,256.81,27.19,0.00),v40,z0,tPen\WObj:=wPaper;
    MoveL Offs(pOrigin,257.55,27.86,0.00),v40,z0,tPen\WObj:=wPaper;
    MoveL Offs(pOrigin,259.50,29.81,0.00),v40,z0,tPen\WObj:=wPaper;
    MoveL Offs(pOrigin,259.77,29.44,0.00),v40,z0,tPen\WObj:=wPaper;
    MoveL Offs(pOrigin,260.41,29.01,0.00),v40,z0,tPen\WObj:=wPaper;
    MoveL Offs(pOrigin,264.66,29.01,0.00),v40,z0,tPen\WObj:=wPaper;
    MoveL Offs(pOrigin,271.04,30.29,0.00),v40,z0,tPen\WObj:=wPaper;
    MoveL Offs(pOrigin,282.30,34.04,0.00),v40,z0,tPen\WObj:=wPaper;
    MoveL Offs(pOrigin,284.42,35.10,0.00),v40,z0,tPen\WObj:=wPaper;
    MoveL Offs(pOrigin,285.70,36.24,0.00),v40,z0,tPen\WObj:=wPaper;
    MoveL Offs(pOrigin,285.70,36.24,0.00),v40,z0,tPen\WObj:=wPaper;
    MoveL Offs(pOrigin,284.85,40.70,0.00),v40,z0,tPen\WObj:=wPaper;
    MoveL Offs(pOrigin,286.12,41.76,0.00),v40,z0,tPen\WObj:=wPaper;
    MoveL Offs(pOrigin,286.98,41.34,0.00),v40,z0,tPen\WObj:=wPaper;
    MoveL Offs(pOrigin,286.55,41.34,0.00),v40,z0,tPen\WObj:=wPaper;
    MoveL Offs(pOrigin,285.27,42.61,0.00),v40,z0,tPen\WObj:=wPaper;
    MoveL Offs(pOrigin,284.64,42.61,0.00),v40,z0,tPen\WObj:=wPaper;
    MoveL Offs(pOrigin,284.42,41.34,0.00),v40,z0,tPen\WObj:=wPaper;
    MoveL Offs(pOrigin,284.85,41.12,0.00),v40,z0,tPen\WObj:=wPaper;
    MoveL Offs(pOrigin,284.41,41.27,0.00),v40,z0,tPen\WObj:=wPaper;
    MoveL Offs(pOrigin,286.21,43.08,0.00),v40,z0,tPen\WObj:=wPaper;
    MoveL Offs(pOrigin,286.96,42.33,0.00),v40,z0,tPen\WObj:=wPaper;
    MoveL Offs(pOrigin,284.85,40.23,0.00),v40,z0,tPen\WObj:=wPaper;
    MoveL Offs(pOrigin,283.73,40.59,0.00),v40,z0,tPen\WObj:=wPaper;
    MoveL Offs(pOrigin,289.44,34.88,0.00),v40,z0,tPen\WObj:=wPaper;
    MoveL Offs(pOrigin,290.49,35.33,0.00),v40,z0,tPen\WObj:=wPaper;
    MoveL Offs(pOrigin,279.22,46.59,0.00),v40,z0,tPen\WObj:=wPaper;
    MoveL Offs(pOrigin,278.88,46.20,0.00),v40,z0,tPen\WObj:=wPaper;
    MoveL Offs(pOrigin,275.57,42.89,0.00),v40,z0,tPen\WObj:=wPaper;
    MoveL Offs(pOrigin,276.09,42.26,0.00),v40,z0,tPen\WObj:=wPaper;
    MoveL Offs(pOrigin,273.83,44.51,0.00),v40,z0,tPen\WObj:=wPaper;
    MoveL Offs(pOrigin,273.78,44.09,0.00),v40,z0,tPen\WObj:=wPaper;
    MoveL Offs(pOrigin,269.57,39.88,0.00),v40,z0,tPen\WObj:=wPaper;
    MoveL Offs(pOrigin,269.95,39.43,0.00),v40,z0,tPen\WObj:=wPaper;
    MoveL Offs(pOrigin,267.85,41.54,0.00),v40,z0,tPen\WObj:=wPaper;
    MoveL Offs(pOrigin,268.90,41.98,0.00),v40,z0,tPen\WObj:=wPaper;
    MoveL Offs(pOrigin,271.15,39.73,0.00),v40,z0,tPen\WObj:=wPaper;
    MoveL Offs(pOrigin,272.05,40.33,0.00),v40,z0,tPen\WObj:=wPaper;
    MoveL Offs(pOrigin,269.79,42.58,0.00),v40,z0,tPen\WObj:=wPaper;
    MoveL Offs(pOrigin,270.78,42.58,0.00),v40,z0,tPen\WObj:=wPaper;
    MoveL Offs(pOrigin,266.57,38.37,0.00),v40,z0,tPen\WObj:=wPaper;
    MoveL Offs(pOrigin,266.96,37.94,0.00),v40,z0,tPen\WObj:=wPaper;
    MoveL Offs(pOrigin,264.86,40.05,0.00),v40,z0,tPen\WObj:=wPaper;
    MoveL Offs(pOrigin,265.90,40.49,0.00),v40,z0,tPen\WObj:=wPaper;
    MoveL Offs(pOrigin,268.16,38.24,0.00),v40,z0,tPen\WObj:=wPaper;
    MoveL Offs(pOrigin,268.90,38.99,0.00),v40,z0,tPen\WObj:=wPaper;
    MoveL Offs(pOrigin,266.80,41.09,0.00),v40,fine,tPen\WObj:=wPaper;
    MoveL Offs(pOrigin,266.80,41.09,6.00),v60,z5,tPen\WObj:=wPaper;
    MoveL Offs(pOrigin,267.85,39.29,6.00),vTravel,z5,tPen\WObj:=wPaper;
    MoveL Offs(pOrigin,267.85,39.29,0.00),v60,z0,tPen\WObj:=wPaper;
    MoveL Offs(pOrigin,265.73,39.29,0.00),v40,fine,tPen\WObj:=wPaper;
    MoveL Offs(pOrigin,265.73,39.29,6.00),v60,z5,tPen\WObj:=wPaper;
    MoveL Offs(pOrigin,267.00,43.89,6.00),vTravel,z5,tPen\WObj:=wPaper;
    MoveL Offs(pOrigin,267.00,43.89,0.00),v60,z0,tPen\WObj:=wPaper;
    MoveL Offs(pOrigin,265.30,46.65,0.00),v40,fine,tPen\WObj:=wPaper;
    MoveL Offs(pOrigin,265.30,46.65,6.00),v60,z5,tPen\WObj:=wPaper;
    MoveL Offs(pOrigin,263.63,48.74,6.00),vTravel,z5,tPen\WObj:=wPaper;
    MoveL Offs(pOrigin,263.63,48.74,0.00),v60,z0,tPen\WObj:=wPaper;
    MoveL Offs(pOrigin,261.38,50.99,0.00),v40,z0,tPen\WObj:=wPaper;
    MoveL Offs(pOrigin,260.63,50.25,0.00),v40,z0,tPen\WObj:=wPaper;
    MoveL Offs(pOrigin,262.73,48.14,0.00),v40,fine,tPen\WObj:=wPaper;
    MoveL Offs(pOrigin,262.73,48.14,6.00),v60,z5,tPen\WObj:=wPaper;
    MoveL Offs(pOrigin,260.94,46.95,6.00),vTravel,z5,tPen\WObj:=wPaper;
    MoveL Offs(pOrigin,260.94,46.95,0.00),v60,z0,tPen\WObj:=wPaper;
    MoveL Offs(pOrigin,258.69,49.20,0.00),v40,z0,tPen\WObj:=wPaper;
    MoveL Offs(pOrigin,257.79,48.61,0.00),v40,z0,tPen\WObj:=wPaper;
    MoveL Offs(pOrigin,260.04,46.35,0.00),v40,fine,tPen\WObj:=wPaper;
    MoveL Offs(pOrigin,260.04,46.35,6.00),v60,z5,tPen\WObj:=wPaper;
    MoveL Offs(pOrigin,255.71,43.22,6.00),vTravel,z5,tPen\WObj:=wPaper;
    MoveL Offs(pOrigin,255.71,43.22,0.00),v60,z0,tPen\WObj:=wPaper;
    MoveL Offs(pOrigin,253.46,45.48,0.00),v40,fine,tPen\WObj:=wPaper;
    MoveL Offs(pOrigin,253.46,45.48,6.00),v60,z5,tPen\WObj:=wPaper;
  ENDPROC

  PROC DrawPart28()
    MoveL Offs(pOrigin,249.71,46.24,6.00),vTravel,z5,tPen\WObj:=wPaper;
    MoveL Offs(pOrigin,249.71,46.24,0.00),v60,z0,tPen\WObj:=wPaper;
    MoveL Offs(pOrigin,247.45,48.49,0.00),v40,z0,tPen\WObj:=wPaper;
    MoveL Offs(pOrigin,246.86,47.59,0.00),v40,z0,tPen\WObj:=wPaper;
    MoveL Offs(pOrigin,248.96,45.49,0.00),v40,z0,tPen\WObj:=wPaper;
    MoveL Offs(pOrigin,248.21,44.74,0.00),v40,z0,tPen\WObj:=wPaper;
    MoveL Offs(pOrigin,245.96,47.00,0.00),v40,z0,tPen\WObj:=wPaper;
    MoveL Offs(pOrigin,245.36,46.10,0.00),v40,z0,tPen\WObj:=wPaper;
    MoveL Offs(pOrigin,247.62,43.85,0.00),v40,z0,tPen\WObj:=wPaper;
    MoveL Offs(pOrigin,247.02,44.57,0.00),v40,z0,tPen\WObj:=wPaper;
    MoveL Offs(pOrigin,245.54,44.57,0.00),v40,z0,tPen\WObj:=wPaper;
    MoveL Offs(pOrigin,245.47,45.65,0.00),v40,z0,tPen\WObj:=wPaper;
    MoveL Offs(pOrigin,258.24,58.42,0.00),v40,z0,tPen\WObj:=wPaper;
    MoveL Offs(pOrigin,258.06,58.79,0.00),v40,z0,tPen\WObj:=wPaper;
    MoveL Offs(pOrigin,260.46,56.39,0.00),v40,z0,tPen\WObj:=wPaper;
    MoveL Offs(pOrigin,261.36,56.99,0.00),v40,z0,tPen\WObj:=wPaper;
    MoveL Offs(pOrigin,258.96,59.39,0.00),v40,z0,tPen\WObj:=wPaper;
    MoveL Offs(pOrigin,259.85,59.99,0.00),v40,z0,tPen\WObj:=wPaper;
    MoveL Offs(pOrigin,262.26,57.58,0.00),v40,fine,tPen\WObj:=wPaper;
    MoveL Offs(pOrigin,262.26,57.58,6.00),v60,z5,tPen\WObj:=wPaper;
    MoveL Offs(pOrigin,262.54,58.97,6.00),vTravel,z5,tPen\WObj:=wPaper;
    MoveL Offs(pOrigin,262.54,58.97,0.00),v60,z0,tPen\WObj:=wPaper;
    MoveL Offs(pOrigin,263.17,59.40,0.00),v40,z0,tPen\WObj:=wPaper;
    MoveL Offs(pOrigin,262.54,58.97,0.00),v40,fine,tPen\WObj:=wPaper;
    MoveL Offs(pOrigin,262.54,58.97,6.00),v60,z5,tPen\WObj:=wPaper;
    MoveL Offs(pOrigin,262.00,60.68,6.00),vTravel,z5,tPen\WObj:=wPaper;
    MoveL Offs(pOrigin,262.00,60.68,0.00),v60,z0,tPen\WObj:=wPaper;
    MoveL Offs(pOrigin,240.06,38.74,0.00),v40,fine,tPen\WObj:=wPaper;
    MoveL Offs(pOrigin,240.06,38.74,6.00),v60,z5,tPen\WObj:=wPaper;
    MoveL Offs(pOrigin,238.56,38.74,6.00),vTravel,z5,tPen\WObj:=wPaper;
    MoveL Offs(pOrigin,238.56,38.74,0.00),v60,z0,tPen\WObj:=wPaper;
    MoveL Offs(pOrigin,240.51,40.69,0.00),v40,z0,tPen\WObj:=wPaper;
    MoveL Offs(pOrigin,239.80,40.34,0.00),v40,z0,tPen\WObj:=wPaper;
    MoveL Offs(pOrigin,218.76,40.34,0.00),v40,z0,tPen\WObj:=wPaper;
    MoveL Offs(pOrigin,219.09,40.17,0.00),v40,z0,tPen\WObj:=wPaper;
    MoveL Offs(pOrigin,225.10,46.18,0.00),v40,z0,tPen\WObj:=wPaper;
    MoveL Offs(pOrigin,225.59,46.46,0.00),v40,z0,tPen\WObj:=wPaper;
    MoveL Offs(pOrigin,215.67,56.38,0.00),v40,z0,tPen\WObj:=wPaper;
    MoveL Offs(pOrigin,216.29,56.79,0.00),v40,z0,tPen\WObj:=wPaper;
    MoveL Offs(pOrigin,218.10,58.60,0.00),v40,z0,tPen\WObj:=wPaper;
    MoveL Offs(pOrigin,217.49,58.76,0.00),v40,z0,tPen\WObj:=wPaper;
    MoveL Offs(pOrigin,217.27,59.19,0.00),v40,z0,tPen\WObj:=wPaper;
    MoveL Offs(pOrigin,217.49,58.76,0.00),v40,z0,tPen\WObj:=wPaper;
    MoveL Offs(pOrigin,217.49,58.30,0.00),v40,z0,tPen\WObj:=wPaper;
    MoveL Offs(pOrigin,216.21,58.30,0.00),v40,z0,tPen\WObj:=wPaper;
    MoveL Offs(pOrigin,216.00,57.99,0.00),v40,z0,tPen\WObj:=wPaper;
    MoveL Offs(pOrigin,217.65,59.64,0.00),v40,z0,tPen\WObj:=wPaper;
    MoveL Offs(pOrigin,217.28,59.35,0.00),v40,z0,tPen\WObj:=wPaper;
    MoveL Offs(pOrigin,215.36,59.35,0.00),v40,z0,tPen\WObj:=wPaper;
    MoveL Offs(pOrigin,214.94,59.19,0.00),v40,z0,tPen\WObj:=wPaper;
    MoveL Offs(pOrigin,216.21,58.34,0.00),v40,z0,tPen\WObj:=wPaper;
    MoveL Offs(pOrigin,216.85,56.85,0.00),v40,z0,tPen\WObj:=wPaper;
    MoveL Offs(pOrigin,216.85,56.00,0.00),v40,z0,tPen\WObj:=wPaper;
    MoveL Offs(pOrigin,216.28,54.72,0.00),v40,z0,tPen\WObj:=wPaper;
    MoveL Offs(pOrigin,214.94,53.38,0.00),v40,z0,tPen\WObj:=wPaper;
    MoveL Offs(pOrigin,213.88,53.24,0.00),v40,z0,tPen\WObj:=wPaper;
    MoveL Offs(pOrigin,212.81,53.52,0.00),v40,z0,tPen\WObj:=wPaper;
    MoveL Offs(pOrigin,211.96,53.24,0.00),v40,z0,tPen\WObj:=wPaper;
    MoveL Offs(pOrigin,201.34,58.83,0.00),v40,z0,tPen\WObj:=wPaper;
    MoveL Offs(pOrigin,196.02,60.67,0.00),v40,z0,tPen\WObj:=wPaper;
    MoveL Offs(pOrigin,189.44,62.38,0.00),v40,z0,tPen\WObj:=wPaper;
    MoveL Offs(pOrigin,184.76,64.07,0.00),v40,z0,tPen\WObj:=wPaper;
    MoveL Offs(pOrigin,184.34,63.86,0.00),v40,z0,tPen\WObj:=wPaper;
    MoveL Offs(pOrigin,184.34,63.86,0.00),v40,z0,tPen\WObj:=wPaper;
    MoveL Offs(pOrigin,184.98,62.94,0.00),v40,z0,tPen\WObj:=wPaper;
    MoveL Offs(pOrigin,187.52,61.88,0.00),v40,z0,tPen\WObj:=wPaper;
    MoveL Offs(pOrigin,200.06,57.98,0.00),v40,z0,tPen\WObj:=wPaper;
    MoveL Offs(pOrigin,204.52,55.93,0.00),v40,z0,tPen\WObj:=wPaper;
    MoveL Offs(pOrigin,212.81,50.90,0.00),v40,z0,tPen\WObj:=wPaper;
    MoveL Offs(pOrigin,214.51,48.99,0.00),v40,z0,tPen\WObj:=wPaper;
    MoveL Offs(pOrigin,215.15,47.50,0.00),v40,z0,tPen\WObj:=wPaper;
    MoveL Offs(pOrigin,214.65,44.95,0.00),v40,z0,tPen\WObj:=wPaper;
    MoveL Offs(pOrigin,213.88,44.10,0.00),v40,z0,tPen\WObj:=wPaper;
    MoveL Offs(pOrigin,212.18,43.25,0.00),v40,z0,tPen\WObj:=wPaper;
    MoveL Offs(pOrigin,209.41,43.25,0.00),v40,z0,tPen\WObj:=wPaper;
    MoveL Offs(pOrigin,193.90,47.50,0.00),v40,z0,tPen\WObj:=wPaper;
    MoveL Offs(pOrigin,184.34,50.90,0.00),v40,z0,tPen\WObj:=wPaper;
    MoveL Offs(pOrigin,183.77,50.69,0.00),v40,z0,tPen\WObj:=wPaper;
    MoveL Offs(pOrigin,184.34,49.98,0.00),v40,z0,tPen\WObj:=wPaper;
    MoveL Offs(pOrigin,188.52,48.07,0.00),v40,z0,tPen\WObj:=wPaper;
    MoveL Offs(pOrigin,189.44,46.72,0.00),v40,z0,tPen\WObj:=wPaper;
    MoveL Offs(pOrigin,190.50,46.44,0.00),v40,z0,tPen\WObj:=wPaper;
    MoveL Offs(pOrigin,190.50,46.44,0.00),v40,z0,tPen\WObj:=wPaper;
    MoveL Offs(pOrigin,190.07,45.38,0.00),v40,z0,tPen\WObj:=wPaper;
    MoveL Offs(pOrigin,189.30,44.74,0.00),v40,z0,tPen\WObj:=wPaper;
    MoveL Offs(pOrigin,189.51,43.96,0.00),v40,z0,tPen\WObj:=wPaper;
    MoveL Offs(pOrigin,190.29,43.46,0.00),v40,z0,tPen\WObj:=wPaper;
    MoveL Offs(pOrigin,190.29,43.46,0.00),v40,z0,tPen\WObj:=wPaper;
    MoveL Offs(pOrigin,190.71,43.89,0.00),v40,z0,tPen\WObj:=wPaper;
    MoveL Offs(pOrigin,190.71,44.95,0.00),v40,z0,tPen\WObj:=wPaper;
    MoveL Offs(pOrigin,190.29,45.38,0.00),v40,z0,tPen\WObj:=wPaper;
    MoveL Offs(pOrigin,190.29,45.62,0.00),v40,z0,tPen\WObj:=wPaper;
    MoveL Offs(pOrigin,188.38,45.62,0.00),v40,z0,tPen\WObj:=wPaper;
    MoveL Offs(pOrigin,188.80,46.22,0.00),v40,z0,tPen\WObj:=wPaper;
    MoveL Offs(pOrigin,188.80,44.38,0.00),v40,z0,tPen\WObj:=wPaper;
    MoveL Offs(pOrigin,186.68,44.31,0.00),v40,z0,tPen\WObj:=wPaper;
    MoveL Offs(pOrigin,186.68,44.31,0.00),v40,z0,tPen\WObj:=wPaper;
    MoveL Offs(pOrigin,185.82,43.46,0.00),v40,z0,tPen\WObj:=wPaper;
    MoveL Offs(pOrigin,185.82,43.46,0.00),v40,z0,tPen\WObj:=wPaper;
    MoveL Offs(pOrigin,187.31,45.45,0.00),v40,z0,tPen\WObj:=wPaper;
    MoveL Offs(pOrigin,189.23,46.65,0.00),v40,z0,tPen\WObj:=wPaper;
    MoveL Offs(pOrigin,189.01,46.68,0.00),v40,z0,tPen\WObj:=wPaper;
    MoveL Offs(pOrigin,195.39,46.68,0.00),v40,z0,tPen\WObj:=wPaper;
    MoveL Offs(pOrigin,194.99,47.44,0.00),v40,z0,tPen\WObj:=wPaper;
    MoveL Offs(pOrigin,193.64,46.09,0.00),v40,z0,tPen\WObj:=wPaper;
    MoveL Offs(pOrigin,193.99,45.21,0.00),v40,z0,tPen\WObj:=wPaper;
    MoveL Offs(pOrigin,189.48,49.72,0.00),v40,z0,tPen\WObj:=wPaper;
    MoveL Offs(pOrigin,189.46,49.37,0.00),v40,z0,tPen\WObj:=wPaper;
    MoveL Offs(pOrigin,187.80,47.72,0.00),v40,z0,tPen\WObj:=wPaper;
    MoveL Offs(pOrigin,188.59,47.74,0.00),v40,z0,tPen\WObj:=wPaper;
    MoveL Offs(pOrigin,191.99,47.74,0.00),v40,z0,tPen\WObj:=wPaper;
    MoveL Offs(pOrigin,192.75,48.18,0.00),v40,z0,tPen\WObj:=wPaper;
    MoveL Offs(pOrigin,188.69,44.12,0.00),v40,z0,tPen\WObj:=wPaper;
    MoveL Offs(pOrigin,188.59,44.57,0.00),v40,z0,tPen\WObj:=wPaper;
    MoveL Offs(pOrigin,190.50,44.57,0.00),v40,z0,tPen\WObj:=wPaper;
    MoveL Offs(pOrigin,191.09,45.03,0.00),v40,z0,tPen\WObj:=wPaper;
    MoveL Offs(pOrigin,189.59,43.53,0.00),v40,z0,tPen\WObj:=wPaper;
    MoveL Offs(pOrigin,190.29,43.46,0.00),v40,z0,tPen\WObj:=wPaper;
    MoveL Offs(pOrigin,190.50,41.76,0.00),v40,z0,tPen\WObj:=wPaper;
    MoveL Offs(pOrigin,191.07,41.97,0.00),v40,z0,tPen\WObj:=wPaper;
  ENDPROC

  PROC DrawPart29()
    MoveL Offs(pOrigin,191.14,43.04,0.00),v40,z0,tPen\WObj:=wPaper;
    MoveL Offs(pOrigin,190.71,43.46,0.00),v40,z0,tPen\WObj:=wPaper;
    MoveL Offs(pOrigin,191.92,42.61,0.00),v40,z0,tPen\WObj:=wPaper;
    MoveL Offs(pOrigin,191.99,41.12,0.00),v40,z0,tPen\WObj:=wPaper;
    MoveL Offs(pOrigin,191.77,40.70,0.00),v40,z0,tPen\WObj:=wPaper;
    MoveL Offs(pOrigin,190.50,40.06,0.00),v40,z0,tPen\WObj:=wPaper;
    MoveL Offs(pOrigin,190.50,40.06,0.00),v40,z0,tPen\WObj:=wPaper;
    MoveL Offs(pOrigin,189.86,39.21,0.00),v40,z0,tPen\WObj:=wPaper;
    MoveL Offs(pOrigin,189.23,39.42,0.00),v40,z0,tPen\WObj:=wPaper;
    MoveL Offs(pOrigin,189.23,39.21,0.00),v40,z0,tPen\WObj:=wPaper;
    MoveL Offs(pOrigin,189.23,39.21,0.00),v40,z0,tPen\WObj:=wPaper;
    MoveL Offs(pOrigin,188.80,38.65,0.00),v40,z0,tPen\WObj:=wPaper;
    MoveL Offs(pOrigin,187.52,38.58,0.00),v40,z0,tPen\WObj:=wPaper;
    MoveL Offs(pOrigin,187.10,38.79,0.00),v40,z0,tPen\WObj:=wPaper;
    MoveL Offs(pOrigin,186.89,39.42,0.00),v40,z0,tPen\WObj:=wPaper;
    MoveL Offs(pOrigin,186.89,39.42,0.00),v40,z0,tPen\WObj:=wPaper;
    MoveL Offs(pOrigin,189.23,39.21,0.00),v40,z0,tPen\WObj:=wPaper;
    MoveL Offs(pOrigin,190.07,39.21,0.00),v40,z0,tPen\WObj:=wPaper;
    MoveL Offs(pOrigin,190.15,38.36,0.00),v40,z0,tPen\WObj:=wPaper;
    MoveL Offs(pOrigin,190.50,38.01,0.00),v40,z0,tPen\WObj:=wPaper;
    MoveL Offs(pOrigin,195.39,36.88,0.00),v40,z0,tPen\WObj:=wPaper;
    MoveL Offs(pOrigin,199.64,36.88,0.00),v40,z0,tPen\WObj:=wPaper;
    MoveL Offs(pOrigin,203.25,37.87,0.00),v40,z0,tPen\WObj:=wPaper;
    MoveL Offs(pOrigin,205.38,38.93,0.00),v40,z0,tPen\WObj:=wPaper;
    MoveL Offs(pOrigin,207.29,40.28,0.00),v40,z0,tPen\WObj:=wPaper;
    MoveL Offs(pOrigin,208.35,41.76,0.00),v40,z0,tPen\WObj:=wPaper;
    MoveL Offs(pOrigin,208.28,42.12,0.00),v40,z0,tPen\WObj:=wPaper;
    MoveL Offs(pOrigin,191.99,46.86,0.00),v40,z0,tPen\WObj:=wPaper;
    MoveL Offs(pOrigin,190.50,46.44,0.00),v40,fine,tPen\WObj:=wPaper;
    MoveL Offs(pOrigin,190.50,46.44,6.00),v60,z5,tPen\WObj:=wPaper;
    MoveL Offs(pOrigin,192.04,45.66,6.00),vTravel,z5,tPen\WObj:=wPaper;
    MoveL Offs(pOrigin,192.04,45.66,0.00),v60,z0,tPen\WObj:=wPaper;
    MoveL Offs(pOrigin,187.08,50.62,0.00),v40,z0,tPen\WObj:=wPaper;
    MoveL Offs(pOrigin,187.06,49.96,0.00),v40,z0,tPen\WObj:=wPaper;
    MoveL Offs(pOrigin,186.16,49.06,0.00),v40,z0,tPen\WObj:=wPaper;
    MoveL Offs(pOrigin,187.06,48.46,0.00),v40,z0,tPen\WObj:=wPaper;
    MoveL Offs(pOrigin,188.26,49.67,0.00),v40,z0,tPen\WObj:=wPaper;
    MoveL Offs(pOrigin,188.80,48.79,0.00),v40,z0,tPen\WObj:=wPaper;
    MoveL Offs(pOrigin,187.52,48.79,0.00),v40,fine,tPen\WObj:=wPaper;
    MoveL Offs(pOrigin,187.52,48.79,6.00),v60,z5,tPen\WObj:=wPaper;
    MoveL Offs(pOrigin,186.02,50.41,6.00),vTravel,z5,tPen\WObj:=wPaper;
    MoveL Offs(pOrigin,186.02,50.41,0.00),v60,z0,tPen\WObj:=wPaper;
    MoveL Offs(pOrigin,185.11,49.51,0.00),v40,z0,tPen\WObj:=wPaper;
    MoveL Offs(pOrigin,184.39,48.83,0.00),v40,z0,tPen\WObj:=wPaper;
    MoveL Offs(pOrigin,181.23,51.99,0.00),v40,z0,tPen\WObj:=wPaper;
    MoveL Offs(pOrigin,181.15,52.39,0.00),v40,z0,tPen\WObj:=wPaper;
    MoveL Offs(pOrigin,183.70,50.90,0.00),v40,z0,tPen\WObj:=wPaper;
    MoveL Offs(pOrigin,184.22,50.10,0.00),v40,z0,tPen\WObj:=wPaper;
    MoveL Offs(pOrigin,184.97,50.85,0.00),v40,z0,tPen\WObj:=wPaper;
    MoveL Offs(pOrigin,184.68,51.53,0.00),v40,z0,tPen\WObj:=wPaper;
    MoveL Offs(pOrigin,191.74,44.47,0.00),v40,z0,tPen\WObj:=wPaper;
    MoveL Offs(pOrigin,191.39,43.83,0.00),v40,z0,tPen\WObj:=wPaper;
    MoveL Offs(pOrigin,190.34,42.78,0.00),v40,fine,tPen\WObj:=wPaper;
    MoveL Offs(pOrigin,190.34,42.78,6.00),v60,z5,tPen\WObj:=wPaper;
    MoveL Offs(pOrigin,190.63,41.58,6.00),vTravel,z5,tPen\WObj:=wPaper;
    MoveL Offs(pOrigin,190.63,41.58,0.00),v60,z0,tPen\WObj:=wPaper;
    MoveL Offs(pOrigin,191.83,42.79,0.00),v40,z0,tPen\WObj:=wPaper;
    MoveL Offs(pOrigin,192.50,42.22,0.00),v40,z0,tPen\WObj:=wPaper;
    MoveL Offs(pOrigin,182.43,52.28,0.00),v40,fine,tPen\WObj:=wPaper;
    MoveL Offs(pOrigin,182.43,52.28,6.00),v60,z5,tPen\WObj:=wPaper;
    MoveL Offs(pOrigin,186.94,46.28,6.00),vTravel,z5,tPen\WObj:=wPaper;
    MoveL Offs(pOrigin,186.94,46.28,0.00),v60,z0,tPen\WObj:=wPaper;
    MoveL Offs(pOrigin,192.50,40.72,0.00),v40,z0,tPen\WObj:=wPaper;
    MoveL Offs(pOrigin,191.98,41.44,0.00),v40,z0,tPen\WObj:=wPaper;
    MoveL Offs(pOrigin,187.62,37.08,0.00),v40,z0,tPen\WObj:=wPaper;
    MoveL Offs(pOrigin,187.87,36.39,0.00),v40,z0,tPen\WObj:=wPaper;
    MoveL Offs(pOrigin,183.21,41.05,0.00),v40,z0,tPen\WObj:=wPaper;
    MoveL Offs(pOrigin,183.66,42.09,0.00),v40,z0,tPen\WObj:=wPaper;
    MoveL Offs(pOrigin,189.82,35.93,0.00),v40,z0,tPen\WObj:=wPaper;
    MoveL Offs(pOrigin,190.17,36.64,0.00),v40,z0,tPen\WObj:=wPaper;
    MoveL Offs(pOrigin,191.52,37.99,0.00),v40,z0,tPen\WObj:=wPaper;
    MoveL Offs(pOrigin,190.50,38.23,0.00),v40,z0,tPen\WObj:=wPaper;
    MoveL Offs(pOrigin,185.40,38.23,0.00),v40,z0,tPen\WObj:=wPaper;
    MoveL Offs(pOrigin,185.53,37.97,0.00),v40,z0,tPen\WObj:=wPaper;
    MoveL Offs(pOrigin,187.03,39.48,0.00),v40,z0,tPen\WObj:=wPaper;
    MoveL Offs(pOrigin,186.89,39.42,0.00),v40,z0,tPen\WObj:=wPaper;
    MoveL Offs(pOrigin,186.04,40.28,0.00),v40,z0,tPen\WObj:=wPaper;
    MoveL Offs(pOrigin,186.04,40.28,0.00),v40,z0,tPen\WObj:=wPaper;
    MoveL Offs(pOrigin,185.82,43.46,0.00),v40,z0,tPen\WObj:=wPaper;
    MoveL Offs(pOrigin,185.82,43.46,0.00),v40,z0,tPen\WObj:=wPaper;
    MoveL Offs(pOrigin,185.05,43.04,0.00),v40,z0,tPen\WObj:=wPaper;
    MoveL Offs(pOrigin,184.76,40.91,0.00),v40,z0,tPen\WObj:=wPaper;
    MoveL Offs(pOrigin,184.98,40.56,0.00),v40,z0,tPen\WObj:=wPaper;
    MoveL Offs(pOrigin,186.04,40.28,0.00),v40,z0,tPen\WObj:=wPaper;
    MoveL Offs(pOrigin,186.28,40.22,0.00),v40,z0,tPen\WObj:=wPaper;
    MoveL Offs(pOrigin,184.33,38.27,0.00),v40,z0,tPen\WObj:=wPaper;
    MoveL Offs(pOrigin,183.43,38.87,0.00),v40,z0,tPen\WObj:=wPaper;
    MoveL Offs(pOrigin,185.69,41.12,0.00),v40,z0,tPen\WObj:=wPaper;
    MoveL Offs(pOrigin,184.76,40.49,0.00),v40,z0,tPen\WObj:=wPaper;
    MoveL Offs(pOrigin,184.12,39.85,0.00),v40,z0,tPen\WObj:=wPaper;
    MoveL Offs(pOrigin,182.00,40.28,0.00),v40,z0,tPen\WObj:=wPaper;
    MoveL Offs(pOrigin,182.00,40.28,0.00),v40,z0,tPen\WObj:=wPaper;
    MoveL Offs(pOrigin,178.39,41.55,0.00),v40,z0,tPen\WObj:=wPaper;
    MoveL Offs(pOrigin,178.87,40.91,0.00),v40,z0,tPen\WObj:=wPaper;
    MoveL Offs(pOrigin,179.77,40.01,0.00),v40,fine,tPen\WObj:=wPaper;
    MoveL Offs(pOrigin,179.77,40.01,6.00),v60,z5,tPen\WObj:=wPaper;
    MoveL Offs(pOrigin,179.62,41.66,6.00),vTravel,z5,tPen\WObj:=wPaper;
    MoveL Offs(pOrigin,179.62,41.66,0.00),v60,z0,tPen\WObj:=wPaper;
    MoveL Offs(pOrigin,183.07,38.20,0.00),v40,fine,tPen\WObj:=wPaper;
    MoveL Offs(pOrigin,183.07,38.20,6.00),v60,z5,tPen\WObj:=wPaper;
    MoveL Offs(pOrigin,183.91,39.29,6.00),vTravel,z5,tPen\WObj:=wPaper;
    MoveL Offs(pOrigin,183.91,39.29,0.00),v60,z0,tPen\WObj:=wPaper;
    MoveL Offs(pOrigin,186.46,39.29,0.00),v40,fine,tPen\WObj:=wPaper;
    MoveL Offs(pOrigin,186.46,39.29,6.00),v60,z5,tPen\WObj:=wPaper;
    MoveL Offs(pOrigin,185.82,38.15,6.00),vTravel,z5,tPen\WObj:=wPaper;
    MoveL Offs(pOrigin,185.82,38.15,0.00),v60,z0,tPen\WObj:=wPaper;
    MoveL Offs(pOrigin,182.64,39.35,0.00),v40,z0,tPen\WObj:=wPaper;
    MoveL Offs(pOrigin,182.00,40.28,0.00),v40,z0,tPen\WObj:=wPaper;
    MoveL Offs(pOrigin,182.69,39.61,0.00),v40,z0,tPen\WObj:=wPaper;
    MoveL Offs(pOrigin,191.70,48.63,0.00),v40,z0,tPen\WObj:=wPaper;
    MoveL Offs(pOrigin,191.73,48.96,0.00),v40,z0,tPen\WObj:=wPaper;
    MoveL Offs(pOrigin,196.39,44.30,0.00),v40,z0,tPen\WObj:=wPaper;
    MoveL Offs(pOrigin,197.08,45.05,0.00),v40,z0,tPen\WObj:=wPaper;
    MoveL Offs(pOrigin,198.59,46.55,0.00),v40,z0,tPen\WObj:=wPaper;
    MoveL Offs(pOrigin,198.18,46.99,0.00),v40,z0,tPen\WObj:=wPaper;
    MoveL Offs(pOrigin,202.53,42.64,0.00),v40,z0,tPen\WObj:=wPaper;
    MoveL Offs(pOrigin,202.92,43.42,0.00),v40,z0,tPen\WObj:=wPaper;
    MoveL Offs(pOrigin,204.27,44.77,0.00),v40,z0,tPen\WObj:=wPaper;
    MoveL Offs(pOrigin,204.32,45.33,0.00),v40,z0,tPen\WObj:=wPaper;
    MoveL Offs(pOrigin,210.03,39.62,0.00),v40,z0,tPen\WObj:=wPaper;
  ENDPROC

  PROC DrawPart30()
    MoveL Offs(pOrigin,209.62,40.34,0.00),v40,z0,tPen\WObj:=wPaper;
    MoveL Offs(pOrigin,207.71,40.34,0.00),v40,z0,tPen\WObj:=wPaper;
    MoveL Offs(pOrigin,207.50,40.28,0.00),v40,z0,tPen\WObj:=wPaper;
    MoveL Offs(pOrigin,208.14,40.91,0.00),v40,z0,tPen\WObj:=wPaper;
    MoveL Offs(pOrigin,207.50,40.28,0.00),v40,fine,tPen\WObj:=wPaper;
    MoveL Offs(pOrigin,207.50,40.28,6.00),v60,z5,tPen\WObj:=wPaper;
    MoveL Offs(pOrigin,208.35,39.42,6.00),vTravel,z5,tPen\WObj:=wPaper;
    MoveL Offs(pOrigin,208.35,39.42,0.00),v60,z0,tPen\WObj:=wPaper;
    MoveL Offs(pOrigin,209.20,40.06,0.00),v40,z0,tPen\WObj:=wPaper;
    MoveL Offs(pOrigin,208.35,39.42,0.00),v40,z0,tPen\WObj:=wPaper;
    MoveL Offs(pOrigin,208.35,39.29,0.00),v40,z0,tPen\WObj:=wPaper;
    MoveL Offs(pOrigin,206.44,39.29,0.00),v40,z0,tPen\WObj:=wPaper;
    MoveL Offs(pOrigin,206.28,40.38,0.00),v40,z0,tPen\WObj:=wPaper;
    MoveL Offs(pOrigin,208.39,38.27,0.00),v40,z0,tPen\WObj:=wPaper;
    MoveL Offs(pOrigin,207.71,38.79,0.00),v40,z0,tPen\WObj:=wPaper;
    MoveL Offs(pOrigin,208.14,39.21,0.00),v40,z0,tPen\WObj:=wPaper;
    MoveL Offs(pOrigin,207.71,38.79,0.00),v40,fine,tPen\WObj:=wPaper;
    MoveL Offs(pOrigin,207.71,38.79,6.00),v60,z5,tPen\WObj:=wPaper;
    MoveL Offs(pOrigin,207.64,37.53,6.00),vTravel,z5,tPen\WObj:=wPaper;
    MoveL Offs(pOrigin,207.64,37.53,0.00),v60,z0,tPen\WObj:=wPaper;
    MoveL Offs(pOrigin,205.39,39.78,0.00),v40,z0,tPen\WObj:=wPaper;
    MoveL Offs(pOrigin,204.34,39.33,0.00),v40,z0,tPen\WObj:=wPaper;
    MoveL Offs(pOrigin,206.74,36.93,0.00),v40,fine,tPen\WObj:=wPaper;
    MoveL Offs(pOrigin,206.74,36.93,6.00),v60,z5,tPen\WObj:=wPaper;
    MoveL Offs(pOrigin,203.68,36.12,6.00),vTravel,z5,tPen\WObj:=wPaper;
    MoveL Offs(pOrigin,203.68,36.12,0.00),v60,z0,tPen\WObj:=wPaper;
    MoveL Offs(pOrigin,193.26,36.12,0.00),v40,z0,tPen\WObj:=wPaper;
    MoveL Offs(pOrigin,193.61,35.60,0.00),v40,z0,tPen\WObj:=wPaper;
    MoveL Offs(pOrigin,195.11,37.10,0.00),v40,z0,tPen\WObj:=wPaper;
    MoveL Offs(pOrigin,195.51,37.71,0.00),v40,z0,tPen\WObj:=wPaper;
    MoveL Offs(pOrigin,201.22,32.00,0.00),v40,z0,tPen\WObj:=wPaper;
    MoveL Offs(pOrigin,201.39,32.93,0.00),v40,z0,tPen\WObj:=wPaper;
    MoveL Offs(pOrigin,202.14,33.68,0.00),v40,fine,tPen\WObj:=wPaper;
    MoveL Offs(pOrigin,202.14,33.68,6.00),v60,z5,tPen\WObj:=wPaper;
    MoveL Offs(pOrigin,203.04,34.58,6.00),vTravel,z5,tPen\WObj:=wPaper;
    MoveL Offs(pOrigin,203.04,34.58,0.00),v60,z0,tPen\WObj:=wPaper;
    MoveL Offs(pOrigin,212.66,44.20,0.00),v40,z0,tPen\WObj:=wPaper;
    MoveL Offs(pOrigin,212.56,44.55,0.00),v40,z0,tPen\WObj:=wPaper;
    MoveL Offs(pOrigin,217.37,39.74,0.00),v40,z0,tPen\WObj:=wPaper;
    MoveL Offs(pOrigin,217.74,40.32,0.00),v40,z0,tPen\WObj:=wPaper;
    MoveL Offs(pOrigin,224.50,47.08,0.00),v40,z0,tPen\WObj:=wPaper;
    MoveL Offs(pOrigin,224.08,46.68,0.00),v40,z0,tPen\WObj:=wPaper;
    MoveL Offs(pOrigin,222.38,46.68,0.00),v40,z0,tPen\WObj:=wPaper;
    MoveL Offs(pOrigin,221.74,46.79,0.00),v40,z0,tPen\WObj:=wPaper;
    MoveL Offs(pOrigin,222.02,45.38,0.00),v40,z0,tPen\WObj:=wPaper;
    MoveL Offs(pOrigin,223.15,45.02,0.00),v40,z0,tPen\WObj:=wPaper;
    MoveL Offs(pOrigin,223.15,46.22,0.00),v40,z0,tPen\WObj:=wPaper;
    MoveL Offs(pOrigin,221.74,46.79,0.00),v40,z0,tPen\WObj:=wPaper;
    MoveL Offs(pOrigin,221.52,46.86,0.00),v40,z0,tPen\WObj:=wPaper;
    MoveL Offs(pOrigin,221.10,46.86,0.00),v40,z0,tPen\WObj:=wPaper;
    MoveL Offs(pOrigin,220.46,46.08,0.00),v40,z0,tPen\WObj:=wPaper;
    MoveL Offs(pOrigin,220.04,46.01,0.00),v40,z0,tPen\WObj:=wPaper;
    MoveL Offs(pOrigin,219.40,46.44,0.00),v40,z0,tPen\WObj:=wPaper;
    MoveL Offs(pOrigin,219.19,47.08,0.00),v40,z0,tPen\WObj:=wPaper;
    MoveL Offs(pOrigin,219.19,47.08,0.00),v40,z0,tPen\WObj:=wPaper;
    MoveL Offs(pOrigin,221.10,47.15,0.00),v40,z0,tPen\WObj:=wPaper;
    MoveL Offs(pOrigin,220.82,48.35,0.00),v40,z0,tPen\WObj:=wPaper;
    MoveL Offs(pOrigin,217.06,52.10,0.00),v40,z0,tPen\WObj:=wPaper;
    MoveL Offs(pOrigin,214.94,51.89,0.00),v40,z0,tPen\WObj:=wPaper;
    MoveL Offs(pOrigin,214.58,51.33,0.00),v40,z0,tPen\WObj:=wPaper;
    MoveL Offs(pOrigin,216.43,48.99,0.00),v40,z0,tPen\WObj:=wPaper;
    MoveL Offs(pOrigin,216.21,48.79,0.00),v40,z0,tPen\WObj:=wPaper;
    MoveL Offs(pOrigin,214.51,48.79,0.00),v40,z0,tPen\WObj:=wPaper;
    MoveL Offs(pOrigin,214.02,48.55,0.00),v40,z0,tPen\WObj:=wPaper;
    MoveL Offs(pOrigin,215.83,50.35,0.00),v40,z0,tPen\WObj:=wPaper;
    MoveL Offs(pOrigin,215.36,50.05,0.00),v40,z0,tPen\WObj:=wPaper;
    MoveL Offs(pOrigin,214.73,50.90,0.00),v40,z0,tPen\WObj:=wPaper;
    MoveL Offs(pOrigin,215.36,50.05,0.00),v40,z0,tPen\WObj:=wPaper;
    MoveL Offs(pOrigin,215.36,49.85,0.00),v40,z0,tPen\WObj:=wPaper;
    MoveL Offs(pOrigin,213.66,49.85,0.00),v40,z0,tPen\WObj:=wPaper;
    MoveL Offs(pOrigin,213.66,49.84,0.00),v40,z0,tPen\WObj:=wPaper;
    MoveL Offs(pOrigin,212.60,50.90,0.00),v40,z0,tPen\WObj:=wPaper;
    MoveL Offs(pOrigin,213.66,49.84,0.00),v40,z0,tPen\WObj:=wPaper;
    MoveL Offs(pOrigin,213.58,49.59,0.00),v40,z0,tPen\WObj:=wPaper;
    MoveL Offs(pOrigin,218.53,54.55,0.00),v40,z0,tPen\WObj:=wPaper;
    MoveL Offs(pOrigin,218.97,54.57,0.00),v40,z0,tPen\WObj:=wPaper;
    MoveL Offs(pOrigin,201.84,71.70,0.00),v40,z0,tPen\WObj:=wPaper;
    MoveL Offs(pOrigin,202.11,70.98,0.00),v40,z0,tPen\WObj:=wPaper;
    MoveL Offs(pOrigin,200.75,69.63,0.00),v40,z0,tPen\WObj:=wPaper;
    MoveL Offs(pOrigin,201.12,69.91,0.00),v40,z0,tPen\WObj:=wPaper;
    MoveL Offs(pOrigin,203.46,69.91,0.00),v40,z0,tPen\WObj:=wPaper;
    MoveL Offs(pOrigin,203.15,70.53,0.00),v40,z0,tPen\WObj:=wPaper;
    MoveL Offs(pOrigin,201.95,69.33,0.00),v40,z0,tPen\WObj:=wPaper;
    MoveL Offs(pOrigin,202.85,68.74,0.00),v40,z0,tPen\WObj:=wPaper;
    MoveL Offs(pOrigin,204.50,70.39,0.00),v40,z0,tPen\WObj:=wPaper;
    MoveL Offs(pOrigin,204.24,70.79,0.00),v40,z0,tPen\WObj:=wPaper;
    MoveL Offs(pOrigin,218.97,56.07,0.00),v40,z0,tPen\WObj:=wPaper;
    MoveL Offs(pOrigin,218.54,56.05,0.00),v40,z0,tPen\WObj:=wPaper;
    MoveL Offs(pOrigin,212.83,50.34,0.00),v40,z0,tPen\WObj:=wPaper;
    MoveL Offs(pOrigin,212.39,50.90,0.00),v40,z0,tPen\WObj:=wPaper;
    MoveL Offs(pOrigin,214.94,50.90,0.00),v40,fine,tPen\WObj:=wPaper;
    MoveL Offs(pOrigin,214.94,50.90,6.00),v60,z5,tPen\WObj:=wPaper;
    MoveL Offs(pOrigin,214.38,49.84,6.00),vTravel,z5,tPen\WObj:=wPaper;
    MoveL Offs(pOrigin,214.38,49.84,0.00),v60,z0,tPen\WObj:=wPaper;
    MoveL Offs(pOrigin,214.38,52.60,0.00),v40,z0,tPen\WObj:=wPaper;
    MoveL Offs(pOrigin,213.33,52.60,0.00),v40,z0,tPen\WObj:=wPaper;
    MoveL Offs(pOrigin,213.33,50.90,0.00),v40,fine,tPen\WObj:=wPaper;
    MoveL Offs(pOrigin,213.33,50.90,6.00),v60,z5,tPen\WObj:=wPaper;
    MoveL Offs(pOrigin,211.93,50.94,6.00),vTravel,z5,tPen\WObj:=wPaper;
    MoveL Offs(pOrigin,211.93,50.94,0.00),v60,z0,tPen\WObj:=wPaper;
    MoveL Offs(pOrigin,218.24,57.25,0.00),v40,z0,tPen\WObj:=wPaper;
    MoveL Offs(pOrigin,217.91,57.24,0.00),v40,z0,tPen\WObj:=wPaper;
    MoveL Offs(pOrigin,216.85,57.24,0.00),v40,z0,tPen\WObj:=wPaper;
    MoveL Offs(pOrigin,216.43,57.70,0.00),v40,z0,tPen\WObj:=wPaper;
    MoveL Offs(pOrigin,216.21,58.12,0.00),v40,z0,tPen\WObj:=wPaper;
    MoveL Offs(pOrigin,216.43,57.70,0.00),v40,fine,tPen\WObj:=wPaper;
    MoveL Offs(pOrigin,216.43,57.70,6.00),v60,z5,tPen\WObj:=wPaper;
    MoveL Offs(pOrigin,216.49,58.98,6.00),vTravel,z5,tPen\WObj:=wPaper;
    MoveL Offs(pOrigin,216.49,58.98,0.00),v60,z0,tPen\WObj:=wPaper;
    MoveL Offs(pOrigin,216.49,68.75,0.00),v40,z0,tPen\WObj:=wPaper;
    MoveL Offs(pOrigin,216.21,68.54,0.00),v40,z0,tPen\WObj:=wPaper;
    MoveL Offs(pOrigin,216.64,68.96,0.00),v40,z0,tPen\WObj:=wPaper;
    MoveL Offs(pOrigin,216.64,80.01,0.00),v40,z0,tPen\WObj:=wPaper;
    MoveL Offs(pOrigin,215.36,93.40,0.00),v40,z0,tPen\WObj:=wPaper;
    MoveL Offs(pOrigin,213.88,101.69,0.00),v40,z0,tPen\WObj:=wPaper;
    MoveL Offs(pOrigin,211.75,110.61,0.00),v40,z0,tPen\WObj:=wPaper;
    MoveL Offs(pOrigin,209.13,119.96,0.00),v40,z0,tPen\WObj:=wPaper;
    MoveL Offs(pOrigin,208.14,120.60,0.00),v40,z0,tPen\WObj:=wPaper;
    MoveL Offs(pOrigin,208.14,120.60,0.00),v40,z0,tPen\WObj:=wPaper;
    MoveL Offs(pOrigin,207.71,123.36,0.00),v40,z0,tPen\WObj:=wPaper;
  ENDPROC

  PROC DrawPart31()
    MoveL Offs(pOrigin,206.86,125.28,0.00),v40,z0,tPen\WObj:=wPaper;
    MoveL Offs(pOrigin,205.59,132.50,0.00),v40,z0,tPen\WObj:=wPaper;
    MoveL Offs(pOrigin,200.27,151.62,0.00),v40,z0,tPen\WObj:=wPaper;
    MoveL Offs(pOrigin,193.69,177.34,0.00),v40,z0,tPen\WObj:=wPaper;
    MoveL Offs(pOrigin,194.11,177.98,0.00),v40,z0,tPen\WObj:=wPaper;
    MoveL Offs(pOrigin,206.58,184.77,0.00),v40,z0,tPen\WObj:=wPaper;
    MoveL Offs(pOrigin,206.44,185.41,0.00),v40,z0,tPen\WObj:=wPaper;
    MoveL Offs(pOrigin,197.09,188.74,0.00),v40,z0,tPen\WObj:=wPaper;
    MoveL Offs(pOrigin,196.24,189.66,0.00),v40,z0,tPen\WObj:=wPaper;
    MoveL Offs(pOrigin,209.20,204.96,0.00),v40,z0,tPen\WObj:=wPaper;
    MoveL Offs(pOrigin,209.62,206.02,0.00),v40,z0,tPen\WObj:=wPaper;
    MoveL Offs(pOrigin,209.62,206.02,0.00),v40,z0,tPen\WObj:=wPaper;
    MoveL Offs(pOrigin,201.34,204.96,0.00),v40,z0,tPen\WObj:=wPaper;
    MoveL Offs(pOrigin,191.56,201.77,0.00),v40,z0,tPen\WObj:=wPaper;
    MoveL Offs(pOrigin,191.56,201.77,0.00),v40,z0,tPen\WObj:=wPaper;
    MoveL Offs(pOrigin,191.35,201.35,0.00),v40,z0,tPen\WObj:=wPaper;
    MoveL Offs(pOrigin,190.50,201.35,0.00),v40,z0,tPen\WObj:=wPaper;
    MoveL Offs(pOrigin,190.50,201.35,0.00),v40,z0,tPen\WObj:=wPaper;
    MoveL Offs(pOrigin,190.57,201.99,0.00),v40,z0,tPen\WObj:=wPaper;
    MoveL Offs(pOrigin,191.77,202.70,0.00),v40,z0,tPen\WObj:=wPaper;
    MoveL Offs(pOrigin,197.51,204.96,0.00),v40,z0,tPen\WObj:=wPaper;
    MoveL Offs(pOrigin,202.61,206.24,0.00),v40,z0,tPen\WObj:=wPaper;
    MoveL Offs(pOrigin,207.07,206.88,0.00),v40,z0,tPen\WObj:=wPaper;
    MoveL Offs(pOrigin,210.69,208.01,0.00),v40,z0,tPen\WObj:=wPaper;
    MoveL Offs(pOrigin,213.88,210.27,0.00),v40,z0,tPen\WObj:=wPaper;
    MoveL Offs(pOrigin,215.01,211.98,0.00),v40,z0,tPen\WObj:=wPaper;
    MoveL Offs(pOrigin,213.88,212.19,0.00),v40,z0,tPen\WObj:=wPaper;
    MoveL Offs(pOrigin,208.35,211.34,0.00),v40,z0,tPen\WObj:=wPaper;
    MoveL Offs(pOrigin,202.19,209.71,0.00),v40,z0,tPen\WObj:=wPaper;
    MoveL Offs(pOrigin,196.02,207.02,0.00),v40,z0,tPen\WObj:=wPaper;
    MoveL Offs(pOrigin,185.61,201.49,0.00),v40,z0,tPen\WObj:=wPaper;
    MoveL Offs(pOrigin,178.39,198.30,0.00),v40,z0,tPen\WObj:=wPaper;
    MoveL Offs(pOrigin,167.12,194.12,0.00),v40,z0,tPen\WObj:=wPaper;
    MoveL Offs(pOrigin,146.94,188.03,0.00),v40,z0,tPen\WObj:=wPaper;
    MoveL Offs(pOrigin,145.88,187.54,0.00),v40,z0,tPen\WObj:=wPaper;
    MoveL Offs(pOrigin,145.45,186.90,0.00),v40,z0,tPen\WObj:=wPaper;
    MoveL Offs(pOrigin,145.45,181.59,0.00),v40,z0,tPen\WObj:=wPaper;
    MoveL Offs(pOrigin,146.51,175.43,0.00),v40,z0,tPen\WObj:=wPaper;
    MoveL Offs(pOrigin,149.27,165.23,0.00),v40,z0,tPen\WObj:=wPaper;
    MoveL Offs(pOrigin,158.62,135.26,0.00),v40,z0,tPen\WObj:=wPaper;
    MoveL Offs(pOrigin,160.32,127.82,0.00),v40,z0,tPen\WObj:=wPaper;
    MoveL Offs(pOrigin,162.66,111.25,0.00),v40,z0,tPen\WObj:=wPaper;
    MoveL Offs(pOrigin,163.09,110.05,0.00),v40,z0,tPen\WObj:=wPaper;
    MoveL Offs(pOrigin,163.65,110.19,0.00),v40,z0,tPen\WObj:=wPaper;
    MoveL Offs(pOrigin,164.93,113.16,0.00),v40,z0,tPen\WObj:=wPaper;
    MoveL Offs(pOrigin,165.78,113.80,0.00),v40,z0,tPen\WObj:=wPaper;
    MoveL Offs(pOrigin,169.46,119.54,0.00),v40,z0,tPen\WObj:=wPaper;
    MoveL Offs(pOrigin,172.65,123.79,0.00),v40,fine,tPen\WObj:=wPaper;
    MoveL Offs(pOrigin,172.65,123.79,6.00),v60,z5,tPen\WObj:=wPaper;
    MoveL Offs(pOrigin,174.42,123.01,6.00),vTravel,z5,tPen\WObj:=wPaper;
    MoveL Offs(pOrigin,174.42,123.01,0.00),v60,z0,tPen\WObj:=wPaper;
    MoveL Offs(pOrigin,176.08,121.36,0.00),v40,z0,tPen\WObj:=wPaper;
    MoveL Offs(pOrigin,176.67,122.26,0.00),v40,z0,tPen\WObj:=wPaper;
    MoveL Offs(pOrigin,175.02,123.91,0.00),v40,z0,tPen\WObj:=wPaper;
    MoveL Offs(pOrigin,175.62,123.79,0.00),v40,z0,tPen\WObj:=wPaper;
    MoveL Offs(pOrigin,175.84,124.21,0.00),v40,z0,tPen\WObj:=wPaper;
    MoveL Offs(pOrigin,175.62,123.79,0.00),v40,z0,tPen\WObj:=wPaper;
    MoveL Offs(pOrigin,175.62,124.81,0.00),v40,z0,tPen\WObj:=wPaper;
    MoveL Offs(pOrigin,177.42,123.01,0.00),v40,z0,tPen\WObj:=wPaper;
    MoveL Offs(pOrigin,177.40,123.93,0.00),v40,z0,tPen\WObj:=wPaper;
    MoveL Offs(pOrigin,171.69,118.22,0.00),v40,z0,tPen\WObj:=wPaper;
    MoveL Offs(pOrigin,171.44,118.53,0.00),v40,z0,tPen\WObj:=wPaper;
    MoveL Offs(pOrigin,173.24,116.73,0.00),v40,z0,tPen\WObj:=wPaper;
    MoveL Offs(pOrigin,172.50,115.98,0.00),v40,z0,tPen\WObj:=wPaper;
    MoveL Offs(pOrigin,170.69,117.78,0.00),v40,z0,tPen\WObj:=wPaper;
    MoveL Offs(pOrigin,169.94,118.53,0.00),v40,z0,tPen\WObj:=wPaper;
    MoveL Offs(pOrigin,168.74,119.74,0.00),v40,z0,tPen\WObj:=wPaper;
    MoveL Offs(pOrigin,167.99,118.99,0.00),v40,z0,tPen\WObj:=wPaper;
    MoveL Offs(pOrigin,171.90,115.08,0.00),v40,z0,tPen\WObj:=wPaper;
    MoveL Offs(pOrigin,171.23,114.78,0.00),v40,z0,tPen\WObj:=wPaper;
    MoveL Offs(pOrigin,159.81,103.36,0.00),v40,z0,tPen\WObj:=wPaper;
    MoveL Offs(pOrigin,159.90,103.70,0.00),v40,z0,tPen\WObj:=wPaper;
    MoveL Offs(pOrigin,164.36,103.70,0.00),v40,z0,tPen\WObj:=wPaper;
    MoveL Offs(pOrigin,164.76,103.82,0.00),v40,z0,tPen\WObj:=wPaper;
    MoveL Offs(pOrigin,159.50,98.56,0.00),v40,z0,tPen\WObj:=wPaper;
    MoveL Offs(pOrigin,159.37,97.74,0.00),v40,z0,tPen\WObj:=wPaper;
    MoveL Offs(pOrigin,156.97,100.15,0.00),v40,z0,tPen\WObj:=wPaper;
    MoveL Offs(pOrigin,157.86,99.91,0.00),v40,z0,tPen\WObj:=wPaper;
    MoveL Offs(pOrigin,156.05,98.10,0.00),v40,z0,tPen\WObj:=wPaper;
    MoveL Offs(pOrigin,156.68,97.45,0.00),v40,z0,tPen\WObj:=wPaper;
    MoveL Offs(pOrigin,154.12,100.01,0.00),v40,z0,tPen\WObj:=wPaper;
    MoveL Offs(pOrigin,154.41,99.45,0.00),v40,z0,tPen\WObj:=wPaper;
    MoveL Offs(pOrigin,153.21,98.24,0.00),v40,z0,tPen\WObj:=wPaper;
    MoveL Offs(pOrigin,153.31,98.93,0.00),v40,z0,tPen\WObj:=wPaper;
    MoveL Offs(pOrigin,152.89,99.35,0.00),v40,z0,tPen\WObj:=wPaper;
    MoveL Offs(pOrigin,151.40,99.35,0.00),v40,z0,tPen\WObj:=wPaper;
    MoveL Offs(pOrigin,151.40,99.14,0.00),v40,z0,tPen\WObj:=wPaper;
    MoveL Offs(pOrigin,151.40,99.14,0.00),v40,z0,tPen\WObj:=wPaper;
    MoveL Offs(pOrigin,152.04,98.50,0.00),v40,z0,tPen\WObj:=wPaper;
    MoveL Offs(pOrigin,153.74,98.93,0.00),v40,z0,tPen\WObj:=wPaper;
    MoveL Offs(pOrigin,153.74,98.93,0.00),v40,z0,tPen\WObj:=wPaper;
    MoveL Offs(pOrigin,158.20,99.35,0.00),v40,z0,tPen\WObj:=wPaper;
    MoveL Offs(pOrigin,161.18,99.99,0.00),v40,z0,tPen\WObj:=wPaper;
    MoveL Offs(pOrigin,161.18,99.99,0.00),v40,z0,tPen\WObj:=wPaper;
    MoveL Offs(pOrigin,160.89,99.35,0.00),v40,z0,tPen\WObj:=wPaper;
    MoveL Offs(pOrigin,160.11,98.85,0.00),v40,z0,tPen\WObj:=wPaper;
    MoveL Offs(pOrigin,157.56,98.29,0.00),v40,z0,tPen\WObj:=wPaper;
    MoveL Offs(pOrigin,154.38,98.29,0.00),v40,z0,tPen\WObj:=wPaper;
    MoveL Offs(pOrigin,153.74,98.93,0.00),v40,z0,tPen\WObj:=wPaper;
    MoveL Offs(pOrigin,152.91,99.44,0.00),v40,z0,tPen\WObj:=wPaper;
    MoveL Offs(pOrigin,152.01,98.54,0.00),v40,z0,tPen\WObj:=wPaper;
    MoveL Offs(pOrigin,151.40,99.14,0.00),v40,z0,tPen\WObj:=wPaper;
    MoveL Offs(pOrigin,148.00,99.35,0.00),v40,z0,tPen\WObj:=wPaper;
    MoveL Offs(pOrigin,144.81,99.99,0.00),v40,fine,tPen\WObj:=wPaper;
    MoveL Offs(pOrigin,144.81,99.99,6.00),v60,z5,tPen\WObj:=wPaper;
    MoveL Offs(pOrigin,146.63,100.03,6.00),vTravel,z5,tPen\WObj:=wPaper;
    MoveL Offs(pOrigin,146.63,100.03,0.00),v60,z0,tPen\WObj:=wPaper;
    MoveL Offs(pOrigin,148.28,98.38,0.00),v40,fine,tPen\WObj:=wPaper;
    MoveL Offs(pOrigin,148.28,98.38,6.00),v60,z5,tPen\WObj:=wPaper;
    MoveL Offs(pOrigin,148.13,100.03,6.00),vTravel,z5,tPen\WObj:=wPaper;
    MoveL Offs(pOrigin,148.13,100.03,0.00),v60,z0,tPen\WObj:=wPaper;
    MoveL Offs(pOrigin,150.23,97.92,0.00),v40,z0,tPen\WObj:=wPaper;
    MoveL Offs(pOrigin,150.66,98.68,0.00),v40,z0,tPen\WObj:=wPaper;
    MoveL Offs(pOrigin,151.41,99.44,0.00),v40,z0,tPen\WObj:=wPaper;
    MoveL Offs(pOrigin,151.13,100.02,0.00),v40,z0,tPen\WObj:=wPaper;
    MoveL Offs(pOrigin,153.53,97.61,0.00),v40,fine,tPen\WObj:=wPaper;
    MoveL Offs(pOrigin,153.53,97.61,6.00),v60,z5,tPen\WObj:=wPaper;
    MoveL Offs(pOrigin,154.70,98.25,6.00),vTravel,z5,tPen\WObj:=wPaper;
    MoveL Offs(pOrigin,154.70,98.25,0.00),v60,z0,tPen\WObj:=wPaper;
    MoveL Offs(pOrigin,155.91,99.45,0.00),v40,z0,tPen\WObj:=wPaper;
  ENDPROC

  PROC DrawPart32()
    MoveL Offs(pOrigin,155.62,100.00,0.00),v40,z0,tPen\WObj:=wPaper;
    MoveL Offs(pOrigin,158.02,97.60,0.00),v40,z0,tPen\WObj:=wPaper;
    MoveL Offs(pOrigin,157.55,98.11,0.00),v40,z0,tPen\WObj:=wPaper;
    MoveL Offs(pOrigin,159.50,100.06,0.00),v40,z0,tPen\WObj:=wPaper;
    MoveL Offs(pOrigin,159.51,100.59,0.00),v40,z0,tPen\WObj:=wPaper;
    MoveL Offs(pOrigin,184.61,75.50,0.00),v40,z0,tPen\WObj:=wPaper;
    MoveL Offs(pOrigin,184.90,76.17,0.00),v40,z0,tPen\WObj:=wPaper;
    MoveL Offs(pOrigin,186.85,78.12,0.00),v40,z0,tPen\WObj:=wPaper;
    MoveL Offs(pOrigin,187.10,77.30,0.00),v40,z0,tPen\WObj:=wPaper;
    MoveL Offs(pOrigin,177.32,77.30,0.00),v40,z0,tPen\WObj:=wPaper;
    MoveL Offs(pOrigin,177.32,76.25,0.00),v40,z0,tPen\WObj:=wPaper;
    MoveL Offs(pOrigin,175.62,76.25,0.00),v40,z0,tPen\WObj:=wPaper;
    MoveL Offs(pOrigin,175.16,76.89,0.00),v40,z0,tPen\WObj:=wPaper;
    MoveL Offs(pOrigin,165.24,66.97,0.00),v40,z0,tPen\WObj:=wPaper;
    MoveL Offs(pOrigin,165.42,67.80,0.00),v40,z0,tPen\WObj:=wPaper;
    MoveL Offs(pOrigin,166.91,67.80,0.00),v40,z0,tPen\WObj:=wPaper;
    MoveL Offs(pOrigin,167.19,67.43,0.00),v40,z0,tPen\WObj:=wPaper;
    MoveL Offs(pOrigin,181.92,82.15,0.00),v40,z0,tPen\WObj:=wPaper;
    MoveL Offs(pOrigin,181.15,81.93,0.00),v40,z0,tPen\WObj:=wPaper;
    MoveL Offs(pOrigin,180.87,82.70,0.00),v40,z0,tPen\WObj:=wPaper;
    MoveL Offs(pOrigin,179.24,83.70,0.00),v40,z0,tPen\WObj:=wPaper;
    MoveL Offs(pOrigin,178.60,84.76,0.00),v40,z0,tPen\WObj:=wPaper;
    MoveL Offs(pOrigin,177.32,85.11,0.00),v40,z0,tPen\WObj:=wPaper;
    MoveL Offs(pOrigin,177.32,85.11,0.00),v40,z0,tPen\WObj:=wPaper;
    MoveL Offs(pOrigin,176.83,86.32,0.00),v40,z0,tPen\WObj:=wPaper;
    MoveL Offs(pOrigin,175.20,86.81,0.00),v40,z0,tPen\WObj:=wPaper;
    MoveL Offs(pOrigin,175.20,86.81,0.00),v40,z0,tPen\WObj:=wPaper;
    MoveL Offs(pOrigin,175.70,85.18,0.00),v40,z0,tPen\WObj:=wPaper;
    MoveL Offs(pOrigin,177.11,84.90,0.00),v40,z0,tPen\WObj:=wPaper;
    MoveL Offs(pOrigin,177.11,84.90,0.00),v40,z0,tPen\WObj:=wPaper;
    MoveL Offs(pOrigin,177.54,83.62,0.00),v40,z0,tPen\WObj:=wPaper;
    MoveL Offs(pOrigin,178.39,83.41,0.00),v40,z0,tPen\WObj:=wPaper;
    MoveL Offs(pOrigin,178.39,83.41,0.00),v40,z0,tPen\WObj:=wPaper;
    MoveL Offs(pOrigin,178.39,82.56,0.00),v40,z0,tPen\WObj:=wPaper;
    MoveL Offs(pOrigin,179.24,81.71,0.00),v40,z0,tPen\WObj:=wPaper;
    MoveL Offs(pOrigin,179.66,81.71,0.00),v40,z0,tPen\WObj:=wPaper;
    MoveL Offs(pOrigin,179.66,81.71,0.00),v40,z0,tPen\WObj:=wPaper;
    MoveL Offs(pOrigin,179.88,82.99,0.00),v40,z0,tPen\WObj:=wPaper;
    MoveL Offs(pOrigin,180.27,83.50,0.00),v40,z0,tPen\WObj:=wPaper;
    MoveL Offs(pOrigin,177.57,80.79,0.00),v40,z0,tPen\WObj:=wPaper;
    MoveL Offs(pOrigin,177.61,81.15,0.00),v40,z0,tPen\WObj:=wPaper;
    MoveL Offs(pOrigin,165.21,86.18,0.00),v40,z0,tPen\WObj:=wPaper;
    MoveL Offs(pOrigin,167.05,80.44,0.00),v40,z0,tPen\WObj:=wPaper;
    MoveL Offs(pOrigin,169.60,74.91,0.00),v40,z0,tPen\WObj:=wPaper;
    MoveL Offs(pOrigin,170.74,73.28,0.00),v40,z0,tPen\WObj:=wPaper;
    MoveL Offs(pOrigin,171.80,73.43,0.00),v40,z0,tPen\WObj:=wPaper;
    MoveL Offs(pOrigin,176.26,77.32,0.00),v40,z0,tPen\WObj:=wPaper;
    MoveL Offs(pOrigin,179.80,78.53,0.00),v40,z0,tPen\WObj:=wPaper;
    MoveL Offs(pOrigin,179.80,79.16,0.00),v40,z0,tPen\WObj:=wPaper;
    MoveL Offs(pOrigin,177.61,81.15,0.00),v40,z0,tPen\WObj:=wPaper;
    MoveL Offs(pOrigin,177.18,81.36,0.00),v40,z0,tPen\WObj:=wPaper;
    MoveL Offs(pOrigin,163.73,92.55,0.00),v40,z0,tPen\WObj:=wPaper;
    MoveL Offs(pOrigin,163.30,94.46,0.00),v40,z0,tPen\WObj:=wPaper;
    MoveL Offs(pOrigin,163.94,95.67,0.00),v40,z0,tPen\WObj:=wPaper;
    MoveL Offs(pOrigin,164.65,95.31,0.00),v40,z0,tPen\WObj:=wPaper;
    MoveL Offs(pOrigin,165.14,93.61,0.00),v40,z0,tPen\WObj:=wPaper;
    MoveL Offs(pOrigin,167.34,90.64,0.00),v40,z0,tPen\WObj:=wPaper;
    MoveL Offs(pOrigin,177.18,81.36,0.00),v40,z0,tPen\WObj:=wPaper;
    MoveL Offs(pOrigin,177.11,81.53,0.00),v40,z0,tPen\WObj:=wPaper;
    MoveL Offs(pOrigin,179.24,81.53,0.00),v40,z0,tPen\WObj:=wPaper;
    MoveL Offs(pOrigin,179.02,81.71,0.00),v40,z0,tPen\WObj:=wPaper;
    MoveL Offs(pOrigin,178.60,82.14,0.00),v40,z0,tPen\WObj:=wPaper;
    MoveL Offs(pOrigin,179.02,81.71,0.00),v40,z0,tPen\WObj:=wPaper;
    MoveL Offs(pOrigin,179.66,81.71,0.00),v40,z0,tPen\WObj:=wPaper;
    MoveL Offs(pOrigin,180.51,80.65,0.00),v40,z0,tPen\WObj:=wPaper;
    MoveL Offs(pOrigin,181.15,80.65,0.00),v40,z0,tPen\WObj:=wPaper;
    MoveL Offs(pOrigin,181.15,80.65,0.00),v40,z0,tPen\WObj:=wPaper;
    MoveL Offs(pOrigin,181.22,81.71,0.00),v40,z0,tPen\WObj:=wPaper;
    MoveL Offs(pOrigin,181.79,81.85,0.00),v40,z0,tPen\WObj:=wPaper;
    MoveL Offs(pOrigin,185.61,78.74,0.00),v40,z0,tPen\WObj:=wPaper;
    MoveL Offs(pOrigin,185.61,78.74,0.00),v40,z0,tPen\WObj:=wPaper;
    MoveL Offs(pOrigin,186.68,79.80,0.00),v40,z0,tPen\WObj:=wPaper;
    MoveL Offs(pOrigin,186.85,79.62,0.00),v40,z0,tPen\WObj:=wPaper;
    MoveL Offs(pOrigin,189.71,82.48,0.00),v40,z0,tPen\WObj:=wPaper;
    MoveL Offs(pOrigin,189.65,81.93,0.00),v40,z0,tPen\WObj:=wPaper;
    MoveL Offs(pOrigin,189.01,82.56,0.00),v40,z0,tPen\WObj:=wPaper;
    MoveL Offs(pOrigin,189.65,81.93,0.00),v40,z0,tPen\WObj:=wPaper;
    MoveL Offs(pOrigin,189.65,81.53,0.00),v40,z0,tPen\WObj:=wPaper;
    MoveL Offs(pOrigin,187.10,81.53,0.00),v40,z0,tPen\WObj:=wPaper;
    MoveL Offs(pOrigin,186.68,81.71,0.00),v40,z0,tPen\WObj:=wPaper;
    MoveL Offs(pOrigin,187.74,81.29,0.00),v40,z0,tPen\WObj:=wPaper;
    MoveL Offs(pOrigin,188.23,80.65,0.00),v40,z0,tPen\WObj:=wPaper;
    MoveL Offs(pOrigin,188.80,77.96,0.00),v40,z0,tPen\WObj:=wPaper;
    MoveL Offs(pOrigin,190.29,77.75,0.00),v40,z0,tPen\WObj:=wPaper;
    MoveL Offs(pOrigin,191.35,76.40,0.00),v40,z0,tPen\WObj:=wPaper;
    MoveL Offs(pOrigin,193.48,75.27,0.00),v40,z0,tPen\WObj:=wPaper;
    MoveL Offs(pOrigin,195.81,73.43,0.00),v40,z0,tPen\WObj:=wPaper;
    MoveL Offs(pOrigin,195.37,72.79,0.00),v40,z0,tPen\WObj:=wPaper;
    MoveL Offs(pOrigin,195.37,75.97,0.00),v40,z0,tPen\WObj:=wPaper;
    MoveL Offs(pOrigin,195.39,76.25,0.00),v40,z0,tPen\WObj:=wPaper;
    MoveL Offs(pOrigin,190.92,76.25,0.00),v40,z0,tPen\WObj:=wPaper;
    MoveL Offs(pOrigin,191.14,76.40,0.00),v40,z0,tPen\WObj:=wPaper;
    MoveL Offs(pOrigin,190.50,75.97,0.00),v40,z0,tPen\WObj:=wPaper;
    MoveL Offs(pOrigin,188.59,76.61,0.00),v40,z0,tPen\WObj:=wPaper;
    MoveL Offs(pOrigin,188.38,77.46,0.00),v40,z0,tPen\WObj:=wPaper;
    MoveL Offs(pOrigin,188.59,77.89,0.00),v40,z0,tPen\WObj:=wPaper;
    MoveL Offs(pOrigin,187.10,77.25,0.00),v40,z0,tPen\WObj:=wPaper;
    MoveL Offs(pOrigin,185.61,78.74,0.00),v40,z0,tPen\WObj:=wPaper;
    MoveL Offs(pOrigin,185.61,78.74,0.00),v40,z0,tPen\WObj:=wPaper;
    MoveL Offs(pOrigin,186.46,79.38,0.00),v40,z0,tPen\WObj:=wPaper;
    MoveL Offs(pOrigin,186.10,78.87,0.00),v40,z0,tPen\WObj:=wPaper;
    MoveL Offs(pOrigin,183.70,76.47,0.00),v40,z0,tPen\WObj:=wPaper;
    MoveL Offs(pOrigin,182.66,75.95,0.00),v40,z0,tPen\WObj:=wPaper;
    MoveL Offs(pOrigin,161.47,97.14,0.00),v40,z0,tPen\WObj:=wPaper;
    MoveL Offs(pOrigin,161.44,96.02,0.00),v40,z0,tPen\WObj:=wPaper;
    MoveL Offs(pOrigin,164.74,99.33,0.00),v40,z0,tPen\WObj:=wPaper;
    MoveL Offs(pOrigin,164.36,99.48,0.00),v40,z0,tPen\WObj:=wPaper;
    MoveL Offs(pOrigin,162.45,99.48,0.00),v40,z0,tPen\WObj:=wPaper;
    MoveL Offs(pOrigin,161.60,99.17,0.00),v40,z0,tPen\WObj:=wPaper;
    MoveL Offs(pOrigin,164.60,102.17,0.00),v40,z0,tPen\WObj:=wPaper;
    MoveL Offs(pOrigin,165.05,102.52,0.00),v40,z0,tPen\WObj:=wPaper;
    MoveL Offs(pOrigin,160.69,106.88,0.00),v40,z0,tPen\WObj:=wPaper;
    MoveL Offs(pOrigin,161.32,106.36,0.00),v40,z0,tPen\WObj:=wPaper;
    MoveL Offs(pOrigin,165.68,110.71,0.00),v40,z0,tPen\WObj:=wPaper;
    MoveL Offs(pOrigin,165.00,111.25,0.00),v40,z0,tPen\WObj:=wPaper;
    MoveL Offs(pOrigin,165.21,111.68,0.00),v40,z0,tPen\WObj:=wPaper;
    MoveL Offs(pOrigin,165.00,111.25,0.00),v40,z0,tPen\WObj:=wPaper;
    MoveL Offs(pOrigin,164.36,111.68,0.00),v40,z0,tPen\WObj:=wPaper;
    MoveL Offs(pOrigin,164.57,112.10,0.00),v40,z0,tPen\WObj:=wPaper;
    MoveL Offs(pOrigin,164.36,111.68,0.00),v40,fine,tPen\WObj:=wPaper;
  ENDPROC

  PROC DrawPart33()
    MoveL Offs(pOrigin,164.36,111.68,6.00),v60,z5,tPen\WObj:=wPaper;
    MoveL Offs(pOrigin,163.14,112.65,6.00),vTravel,z5,tPen\WObj:=wPaper;
    MoveL Offs(pOrigin,163.14,112.65,0.00),v60,z0,tPen\WObj:=wPaper;
    MoveL Offs(pOrigin,160.43,109.95,0.00),v40,z0,tPen\WObj:=wPaper;
    MoveL Offs(pOrigin,160.96,110.04,0.00),v40,z0,tPen\WObj:=wPaper;
    MoveL Offs(pOrigin,164.36,110.04,0.00),v40,z0,tPen\WObj:=wPaper;
    MoveL Offs(pOrigin,164.15,108.98,0.00),v40,z0,tPen\WObj:=wPaper;
    MoveL Offs(pOrigin,161.39,108.98,0.00),v40,z0,tPen\WObj:=wPaper;
    MoveL Offs(pOrigin,160.88,108.90,0.00),v40,z0,tPen\WObj:=wPaper;
    MoveL Offs(pOrigin,167.79,115.81,0.00),v40,fine,tPen\WObj:=wPaper;
    MoveL Offs(pOrigin,167.79,115.81,6.00),v60,z5,tPen\WObj:=wPaper;
    MoveL Offs(pOrigin,165.99,115.51,6.00),vTravel,z5,tPen\WObj:=wPaper;
    MoveL Offs(pOrigin,165.99,115.51,0.00),v60,z0,tPen\WObj:=wPaper;
    MoveL Offs(pOrigin,168.85,118.36,0.00),v40,fine,tPen\WObj:=wPaper;
    MoveL Offs(pOrigin,168.85,118.36,6.00),v60,z5,tPen\WObj:=wPaper;
    MoveL Offs(pOrigin,167.25,118.24,6.00),vTravel,z5,tPen\WObj:=wPaper;
    MoveL Offs(pOrigin,167.25,118.24,0.00),v60,z0,tPen\WObj:=wPaper;
    MoveL Offs(pOrigin,171.30,114.19,0.00),v40,z0,tPen\WObj:=wPaper;
    MoveL Offs(pOrigin,170.71,113.29,0.00),v40,z0,tPen\WObj:=wPaper;
    MoveL Offs(pOrigin,166.65,117.35,0.00),v40,z0,tPen\WObj:=wPaper;
    MoveL Offs(pOrigin,166.05,116.45,0.00),v40,z0,tPen\WObj:=wPaper;
    MoveL Offs(pOrigin,169.96,112.54,0.00),v40,z0,tPen\WObj:=wPaper;
    MoveL Offs(pOrigin,169.52,111.49,0.00),v40,z0,tPen\WObj:=wPaper;
    MoveL Offs(pOrigin,165.46,115.55,0.00),v40,z0,tPen\WObj:=wPaper;
    MoveL Offs(pOrigin,164.86,114.65,0.00),v40,z0,tPen\WObj:=wPaper;
    MoveL Offs(pOrigin,168.77,110.75,0.00),v40,z0,tPen\WObj:=wPaper;
    MoveL Offs(pOrigin,168.17,109.85,0.00),v40,z0,tPen\WObj:=wPaper;
    MoveL Offs(pOrigin,164.27,113.76,0.00),v40,fine,tPen\WObj:=wPaper;
    MoveL Offs(pOrigin,164.27,113.76,6.00),v60,z5,tPen\WObj:=wPaper;
    MoveL Offs(pOrigin,162.84,113.85,6.00),vTravel,z5,tPen\WObj:=wPaper;
    MoveL Offs(pOrigin,162.84,113.85,0.00),v60,z0,tPen\WObj:=wPaper;
    MoveL Offs(pOrigin,159.08,110.10,0.00),v40,z0,tPen\WObj:=wPaper;
    MoveL Offs(pOrigin,159.26,110.82,0.00),v40,z0,tPen\WObj:=wPaper;
    MoveL Offs(pOrigin,143.96,112.53,0.00),v40,z0,tPen\WObj:=wPaper;
    MoveL Offs(pOrigin,139.71,112.31,0.00),v40,z0,tPen\WObj:=wPaper;
    MoveL Offs(pOrigin,139.71,112.31,0.00),v40,z0,tPen\WObj:=wPaper;
    MoveL Offs(pOrigin,140.35,111.68,0.00),v40,z0,tPen\WObj:=wPaper;
    MoveL Offs(pOrigin,146.09,111.46,0.00),v40,z0,tPen\WObj:=wPaper;
    MoveL Offs(pOrigin,156.71,110.19,0.00),v40,z0,tPen\WObj:=wPaper;
    MoveL Offs(pOrigin,158.62,110.19,0.00),v40,z0,tPen\WObj:=wPaper;
    MoveL Offs(pOrigin,159.26,110.82,0.00),v40,z0,tPen\WObj:=wPaper;
    MoveL Offs(pOrigin,159.26,110.82,0.00),v40,z0,tPen\WObj:=wPaper;
    MoveL Offs(pOrigin,159.26,110.61,0.00),v40,z0,tPen\WObj:=wPaper;
    MoveL Offs(pOrigin,160.96,110.82,0.00),v40,z0,tPen\WObj:=wPaper;
    MoveL Offs(pOrigin,160.96,110.82,0.00),v40,z0,tPen\WObj:=wPaper;
    MoveL Offs(pOrigin,160.96,111.89,0.00),v40,z0,tPen\WObj:=wPaper;
    MoveL Offs(pOrigin,160.32,113.38,0.00),v40,z0,tPen\WObj:=wPaper;
    MoveL Offs(pOrigin,158.41,114.93,0.00),v40,z0,tPen\WObj:=wPaper;
    MoveL Offs(pOrigin,154.38,116.14,0.00),v40,z0,tPen\WObj:=wPaper;
    MoveL Offs(pOrigin,150.55,116.14,0.00),v40,z0,tPen\WObj:=wPaper;
    MoveL Offs(pOrigin,148.43,115.71,0.00),v40,z0,tPen\WObj:=wPaper;
    MoveL Offs(pOrigin,147.36,115.93,0.00),v40,z0,tPen\WObj:=wPaper;
    MoveL Offs(pOrigin,147.36,115.93,0.00),v40,z0,tPen\WObj:=wPaper;
    MoveL Offs(pOrigin,148.00,116.56,0.00),v40,z0,tPen\WObj:=wPaper;
    MoveL Offs(pOrigin,151.40,117.20,0.00),v40,z0,tPen\WObj:=wPaper;
    MoveL Offs(pOrigin,155.44,117.20,0.00),v40,z0,tPen\WObj:=wPaper;
    MoveL Offs(pOrigin,160.25,115.93,0.00),v40,z0,tPen\WObj:=wPaper;
    MoveL Offs(pOrigin,160.32,117.62,0.00),v40,z0,tPen\WObj:=wPaper;
    MoveL Offs(pOrigin,159.40,122.51,0.00),v40,z0,tPen\WObj:=wPaper;
    MoveL Offs(pOrigin,156.50,125.49,0.00),v40,z0,tPen\WObj:=wPaper;
    MoveL Offs(pOrigin,156.13,125.07,0.00),v40,z0,tPen\WObj:=wPaper;
    MoveL Offs(pOrigin,160.19,129.12,0.00),v40,z0,tPen\WObj:=wPaper;
    MoveL Offs(pOrigin,159.90,129.05,0.00),v40,z0,tPen\WObj:=wPaper;
    MoveL Offs(pOrigin,156.93,129.05,0.00),v40,z0,tPen\WObj:=wPaper;
    MoveL Offs(pOrigin,156.93,128.68,0.00),v40,z0,tPen\WObj:=wPaper;
    MoveL Offs(pOrigin,156.71,129.10,0.00),v40,z0,tPen\WObj:=wPaper;
    MoveL Offs(pOrigin,156.93,128.68,0.00),v40,z0,tPen\WObj:=wPaper;
    MoveL Offs(pOrigin,157.35,128.46,0.00),v40,z0,tPen\WObj:=wPaper;
    MoveL Offs(pOrigin,157.56,128.04,0.00),v40,z0,tPen\WObj:=wPaper;
    MoveL Offs(pOrigin,157.35,128.46,0.00),v40,z0,tPen\WObj:=wPaper;
    MoveL Offs(pOrigin,157.56,127.99,0.00),v40,z0,tPen\WObj:=wPaper;
    MoveL Offs(pOrigin,160.11,127.99,0.00),v40,z0,tPen\WObj:=wPaper;
    MoveL Offs(pOrigin,160.49,127.93,0.00),v40,z0,tPen\WObj:=wPaper;
    MoveL Offs(pOrigin,157.03,124.47,0.00),v40,z0,tPen\WObj:=wPaper;
    MoveL Offs(pOrigin,157.35,124.43,0.00),v40,z0,tPen\WObj:=wPaper;
    MoveL Offs(pOrigin,157.14,124.85,0.00),v40,z0,tPen\WObj:=wPaper;
    MoveL Offs(pOrigin,157.35,124.43,0.00),v40,z0,tPen\WObj:=wPaper;
    MoveL Offs(pOrigin,157.35,124.82,0.00),v40,z0,tPen\WObj:=wPaper;
    MoveL Offs(pOrigin,160.75,124.82,0.00),v40,z0,tPen\WObj:=wPaper;
    MoveL Offs(pOrigin,160.93,125.38,0.00),v40,z0,tPen\WObj:=wPaper;
    MoveL Offs(pOrigin,158.37,122.83,0.00),v40,z0,tPen\WObj:=wPaper;
    MoveL Offs(pOrigin,159.05,122.94,0.00),v40,z0,tPen\WObj:=wPaper;
    MoveL Offs(pOrigin,159.26,122.51,0.00),v40,z0,tPen\WObj:=wPaper;
    MoveL Offs(pOrigin,159.05,122.94,0.00),v40,z0,tPen\WObj:=wPaper;
    MoveL Offs(pOrigin,159.05,122.71,0.00),v40,z0,tPen\WObj:=wPaper;
    MoveL Offs(pOrigin,160.96,122.71,0.00),v40,z0,tPen\WObj:=wPaper;
    MoveL Offs(pOrigin,161.22,122.69,0.00),v40,z0,tPen\WObj:=wPaper;
    MoveL Offs(pOrigin,159.27,120.73,0.00),v40,z0,tPen\WObj:=wPaper;
    MoveL Offs(pOrigin,158.70,120.82,0.00),v40,z0,tPen\WObj:=wPaper;
    MoveL Offs(pOrigin,162.76,116.76,0.00),v40,z0,tPen\WObj:=wPaper;
    MoveL Offs(pOrigin,162.40,116.40,0.00),v40,z0,tPen\WObj:=wPaper;
    MoveL Offs(pOrigin,159.54,113.54,0.00),v40,z0,tPen\WObj:=wPaper;
    MoveL Offs(pOrigin,159.90,113.59,0.00),v40,z0,tPen\WObj:=wPaper;
    MoveL Offs(pOrigin,159.26,114.22,0.00),v40,z0,tPen\WObj:=wPaper;
    MoveL Offs(pOrigin,159.90,113.59,0.00),v40,z0,tPen\WObj:=wPaper;
    MoveL Offs(pOrigin,160.11,113.21,0.00),v40,z0,tPen\WObj:=wPaper;
    MoveL Offs(pOrigin,162.45,113.21,0.00),v40,z0,tPen\WObj:=wPaper;
    MoveL Offs(pOrigin,162.24,114.26,0.00),v40,z0,tPen\WObj:=wPaper;
    MoveL Offs(pOrigin,159.05,114.26,0.00),v40,z0,tPen\WObj:=wPaper;
    MoveL Offs(pOrigin,158.65,114.14,0.00),v40,z0,tPen\WObj:=wPaper;
    MoveL Offs(pOrigin,162.10,117.59,0.00),v40,z0,tPen\WObj:=wPaper;
    MoveL Offs(pOrigin,161.81,117.43,0.00),v40,z0,tPen\WObj:=wPaper;
    MoveL Offs(pOrigin,160.32,117.43,0.00),v40,z0,tPen\WObj:=wPaper;
    MoveL Offs(pOrigin,159.56,118.04,0.00),v40,z0,tPen\WObj:=wPaper;
    MoveL Offs(pOrigin,161.66,120.14,0.00),v40,z0,tPen\WObj:=wPaper;
    MoveL Offs(pOrigin,162.15,120.36,0.00),v40,z0,tPen\WObj:=wPaper;
    MoveL Offs(pOrigin,145.17,137.33,0.00),v40,z0,tPen\WObj:=wPaper;
    MoveL Offs(pOrigin,145.23,136.57,0.00),v40,z0,tPen\WObj:=wPaper;
    MoveL Offs(pOrigin,144.33,135.67,0.00),v40,z0,tPen\WObj:=wPaper;
    MoveL Offs(pOrigin,144.73,134.79,0.00),v40,z0,tPen\WObj:=wPaper;
    MoveL Offs(pOrigin,141.27,138.25,0.00),v40,z0,tPen\WObj:=wPaper;
    MoveL Offs(pOrigin,141.64,137.46,0.00),v40,z0,tPen\WObj:=wPaper;
    MoveL Offs(pOrigin,140.89,136.70,0.00),v40,z0,tPen\WObj:=wPaper;
    MoveL Offs(pOrigin,140.53,136.00,0.00),v40,z0,tPen\WObj:=wPaper;
    MoveL Offs(pOrigin,138.12,138.41,0.00),v40,fine,tPen\WObj:=wPaper;
    MoveL Offs(pOrigin,138.12,138.41,6.00),v60,z5,tPen\WObj:=wPaper;
    MoveL Offs(pOrigin,139.62,138.40,6.00),vTravel,z5,tPen\WObj:=wPaper;
    MoveL Offs(pOrigin,139.62,138.40,0.00),v60,z0,tPen\WObj:=wPaper;
    MoveL Offs(pOrigin,142.63,135.40,0.00),v40,z0,tPen\WObj:=wPaper;
    MoveL Offs(pOrigin,143.29,136.11,0.00),v40,z0,tPen\WObj:=wPaper;
  ENDPROC

  PROC DrawPart34()
    MoveL Offs(pOrigin,144.19,137.01,0.00),v40,z0,tPen\WObj:=wPaper;
    MoveL Offs(pOrigin,143.75,136.75,0.00),v40,z0,tPen\WObj:=wPaper;
    MoveL Offs(pOrigin,136.95,137.81,0.00),v40,z0,tPen\WObj:=wPaper;
    MoveL Offs(pOrigin,133.55,137.81,0.00),v40,fine,tPen\WObj:=wPaper;
    MoveL Offs(pOrigin,133.55,137.81,6.00),v60,z5,tPen\WObj:=wPaper;
    MoveL Offs(pOrigin,135.43,138.11,6.00),vTravel,z5,tPen\WObj:=wPaper;
    MoveL Offs(pOrigin,135.43,138.11,0.00),v60,z0,tPen\WObj:=wPaper;
    MoveL Offs(pOrigin,136.63,136.91,0.00),v40,fine,tPen\WObj:=wPaper;
    MoveL Offs(pOrigin,136.63,136.91,6.00),v60,z5,tPen\WObj:=wPaper;
    MoveL Offs(pOrigin,136.63,138.41,6.00),vTravel,z5,tPen\WObj:=wPaper;
    MoveL Offs(pOrigin,136.63,138.41,0.00),v60,z0,tPen\WObj:=wPaper;
    MoveL Offs(pOrigin,138.58,136.46,0.00),v40,fine,tPen\WObj:=wPaper;
    MoveL Offs(pOrigin,138.58,136.46,6.00),v60,z5,tPen\WObj:=wPaper;
    MoveL Offs(pOrigin,139.50,133.77,6.00),vTravel,z5,tPen\WObj:=wPaper;
    MoveL Offs(pOrigin,139.50,133.77,0.00),v60,z0,tPen\WObj:=wPaper;
    MoveL Offs(pOrigin,143.54,132.78,0.00),v40,z0,tPen\WObj:=wPaper;
    MoveL Offs(pOrigin,150.34,130.16,0.00),v40,z0,tPen\WObj:=wPaper;
    MoveL Offs(pOrigin,150.34,130.16,0.00),v40,z0,tPen\WObj:=wPaper;
    MoveL Offs(pOrigin,152.25,129.60,0.00),v40,z0,tPen\WObj:=wPaper;
    MoveL Offs(pOrigin,158.62,125.20,0.00),v40,z0,tPen\WObj:=wPaper;
    MoveL Offs(pOrigin,158.98,125.28,0.00),v40,z0,tPen\WObj:=wPaper;
    MoveL Offs(pOrigin,158.91,126.55,0.00),v40,z0,tPen\WObj:=wPaper;
    MoveL Offs(pOrigin,156.07,129.74,0.00),v40,z0,tPen\WObj:=wPaper;
    MoveL Offs(pOrigin,155.65,130.10,0.00),v40,z0,tPen\WObj:=wPaper;
    MoveL Offs(pOrigin,159.69,130.10,0.00),v40,z0,tPen\WObj:=wPaper;
    MoveL Offs(pOrigin,160.05,130.47,0.00),v40,z0,tPen\WObj:=wPaper;
    MoveL Offs(pOrigin,155.39,125.81,0.00),v40,z0,tPen\WObj:=wPaper;
    MoveL Offs(pOrigin,155.23,126.34,0.00),v40,z0,tPen\WObj:=wPaper;
    MoveL Offs(pOrigin,155.93,125.77,0.00),v40,z0,tPen\WObj:=wPaper;
    MoveL Offs(pOrigin,150.76,129.31,0.00),v40,z0,tPen\WObj:=wPaper;
    MoveL Offs(pOrigin,150.34,130.16,0.00),v40,z0,tPen\WObj:=wPaper;
    MoveL Offs(pOrigin,149.91,130.38,0.00),v40,z0,tPen\WObj:=wPaper;
    MoveL Offs(pOrigin,150.34,130.16,0.00),v40,z0,tPen\WObj:=wPaper;
    MoveL Offs(pOrigin,149.91,130.38,0.00),v40,z0,tPen\WObj:=wPaper;
    MoveL Offs(pOrigin,150.01,130.89,0.00),v40,z0,tPen\WObj:=wPaper;
    MoveL Offs(pOrigin,149.11,129.99,0.00),v40,z0,tPen\WObj:=wPaper;
    MoveL Offs(pOrigin,150.01,129.39,0.00),v40,z0,tPen\WObj:=wPaper;
    MoveL Offs(pOrigin,151.06,130.44,0.00),v40,z0,tPen\WObj:=wPaper;
    MoveL Offs(pOrigin,152.11,130.00,0.00),v40,z0,tPen\WObj:=wPaper;
    MoveL Offs(pOrigin,150.90,128.80,0.00),v40,z0,tPen\WObj:=wPaper;
    MoveL Offs(pOrigin,151.95,128.35,0.00),v40,z0,tPen\WObj:=wPaper;
    MoveL Offs(pOrigin,153.00,129.40,0.00),v40,z0,tPen\WObj:=wPaper;
    MoveL Offs(pOrigin,154.05,128.95,0.00),v40,z0,tPen\WObj:=wPaper;
    MoveL Offs(pOrigin,152.70,127.60,0.00),v40,z0,tPen\WObj:=wPaper;
    MoveL Offs(pOrigin,152.69,126.83,0.00),v40,z0,tPen\WObj:=wPaper;
    MoveL Offs(pOrigin,146.68,132.84,0.00),v40,z0,tPen\WObj:=wPaper;
    MoveL Offs(pOrigin,146.87,132.23,0.00),v40,z0,tPen\WObj:=wPaper;
    MoveL Offs(pOrigin,146.12,131.48,0.00),v40,z0,tPen\WObj:=wPaper;
    MoveL Offs(pOrigin,146.09,130.44,0.00),v40,z0,tPen\WObj:=wPaper;
    MoveL Offs(pOrigin,142.63,133.90,0.00),v40,fine,tPen\WObj:=wPaper;
    MoveL Offs(pOrigin,142.63,133.90,6.00),v60,z5,tPen\WObj:=wPaper;
    MoveL Offs(pOrigin,140.83,134.20,6.00),vTravel,z5,tPen\WObj:=wPaper;
    MoveL Offs(pOrigin,140.83,134.20,0.00),v60,z0,tPen\WObj:=wPaper;
    MoveL Offs(pOrigin,143.54,131.50,0.00),v40,z0,tPen\WObj:=wPaper;
    MoveL Offs(pOrigin,142.94,130.60,0.00),v40,z0,tPen\WObj:=wPaper;
    MoveL Offs(pOrigin,146.85,126.69,0.00),v40,fine,tPen\WObj:=wPaper;
    MoveL Offs(pOrigin,146.85,126.69,6.00),v60,z5,tPen\WObj:=wPaper;
    MoveL Offs(pOrigin,148.80,126.24,6.00),vTravel,z5,tPen\WObj:=wPaper;
    MoveL Offs(pOrigin,148.80,126.24,0.00),v60,z0,tPen\WObj:=wPaper;
    MoveL Offs(pOrigin,145.34,129.69,0.00),v40,z0,tPen\WObj:=wPaper;
    MoveL Offs(pOrigin,145.21,129.08,0.00),v40,z0,tPen\WObj:=wPaper;
    MoveL Offs(pOrigin,144.31,128.18,0.00),v40,z0,tPen\WObj:=wPaper;
    MoveL Offs(pOrigin,144.60,128.89,0.00),v40,z0,tPen\WObj:=wPaper;
    MoveL Offs(pOrigin,144.39,129.24,0.00),v40,z0,tPen\WObj:=wPaper;
    MoveL Offs(pOrigin,137.80,131.23,0.00),v40,z0,tPen\WObj:=wPaper;
    MoveL Offs(pOrigin,129.51,132.93,0.00),v40,z0,tPen\WObj:=wPaper;
    MoveL Offs(pOrigin,125.90,133.35,0.00),v40,z0,tPen\WObj:=wPaper;
    MoveL Offs(pOrigin,124.91,133.77,0.00),v40,z0,tPen\WObj:=wPaper;
    MoveL Offs(pOrigin,124.62,135.05,0.00),v40,z0,tPen\WObj:=wPaper;
    MoveL Offs(pOrigin,125.47,136.75,0.00),v40,z0,tPen\WObj:=wPaper;
    MoveL Offs(pOrigin,127.03,138.45,0.00),v40,z0,tPen\WObj:=wPaper;
    MoveL Offs(pOrigin,127.81,140.36,0.00),v40,z0,tPen\WObj:=wPaper;
    MoveL Offs(pOrigin,127.81,146.10,0.00),v40,z0,tPen\WObj:=wPaper;
    MoveL Offs(pOrigin,128.66,147.80,0.00),v40,z0,tPen\WObj:=wPaper;
    MoveL Offs(pOrigin,130.86,150.56,0.00),v40,z0,tPen\WObj:=wPaper;
    MoveL Offs(pOrigin,131.21,151.84,0.00),v40,z0,tPen\WObj:=wPaper;
    MoveL Offs(pOrigin,131.00,155.88,0.00),v40,z0,tPen\WObj:=wPaper;
    MoveL Offs(pOrigin,131.21,156.73,0.00),v40,z0,tPen\WObj:=wPaper;
    MoveL Offs(pOrigin,131.85,157.79,0.00),v40,z0,tPen\WObj:=wPaper;
    MoveL Offs(pOrigin,134.12,159.91,0.00),v40,z0,tPen\WObj:=wPaper;
    MoveL Offs(pOrigin,134.40,160.76,0.00),v40,z0,tPen\WObj:=wPaper;
    MoveL Offs(pOrigin,134.40,164.80,0.00),v40,z0,tPen\WObj:=wPaper;
    MoveL Offs(pOrigin,134.82,166.07,0.00),v40,z0,tPen\WObj:=wPaper;
    MoveL Offs(pOrigin,135.46,166.07,0.00),v40,z0,tPen\WObj:=wPaper;
    MoveL Offs(pOrigin,137.87,161.82,0.00),v40,z0,tPen\WObj:=wPaper;
    MoveL Offs(pOrigin,140.85,158.21,0.00),v40,z0,tPen\WObj:=wPaper;
    MoveL Offs(pOrigin,146.30,152.97,0.00),v40,z0,tPen\WObj:=wPaper;
    MoveL Offs(pOrigin,147.15,152.90,0.00),v40,z0,tPen\WObj:=wPaper;
    MoveL Offs(pOrigin,147.15,152.90,0.00),v40,z0,tPen\WObj:=wPaper;
    MoveL Offs(pOrigin,147.08,153.75,0.00),v40,z0,tPen\WObj:=wPaper;
    MoveL Offs(pOrigin,142.33,158.64,0.00),v40,z0,tPen\WObj:=wPaper;
    MoveL Offs(pOrigin,139.57,162.04,0.00),v40,z0,tPen\WObj:=wPaper;
    MoveL Offs(pOrigin,137.45,165.30,0.00),v40,z0,tPen\WObj:=wPaper;
    MoveL Offs(pOrigin,136.31,167.99,0.00),v40,z0,tPen\WObj:=wPaper;
    MoveL Offs(pOrigin,136.31,169.26,0.00),v40,z0,tPen\WObj:=wPaper;
    MoveL Offs(pOrigin,137.80,173.09,0.00),v40,z0,tPen\WObj:=wPaper;
    MoveL Offs(pOrigin,138.65,178.19,0.00),v40,z0,tPen\WObj:=wPaper;
    MoveL Offs(pOrigin,140.07,182.86,0.00),v40,z0,tPen\WObj:=wPaper;
    MoveL Offs(pOrigin,141.20,184.77,0.00),v40,z0,tPen\WObj:=wPaper;
    MoveL Offs(pOrigin,142.69,186.26,0.00),v40,z0,tPen\WObj:=wPaper;
    MoveL Offs(pOrigin,143.96,186.97,0.00),v40,z0,tPen\WObj:=wPaper;
    MoveL Offs(pOrigin,144.39,186.69,0.00),v40,z0,tPen\WObj:=wPaper;
    MoveL Offs(pOrigin,144.18,181.80,0.00),v40,z0,tPen\WObj:=wPaper;
    MoveL Offs(pOrigin,144.60,178.40,0.00),v40,z0,tPen\WObj:=wPaper;
    MoveL Offs(pOrigin,146.09,171.60,0.00),v40,z0,tPen\WObj:=wPaper;
    MoveL Offs(pOrigin,148.64,162.89,0.00),v40,z0,tPen\WObj:=wPaper;
    MoveL Offs(pOrigin,148.57,162.04,0.00),v40,z0,tPen\WObj:=wPaper;
    MoveL Offs(pOrigin,148.21,161.82,0.00),v40,z0,tPen\WObj:=wPaper;
    MoveL Offs(pOrigin,148.21,161.82,0.00),v40,z0,tPen\WObj:=wPaper;
    MoveL Offs(pOrigin,150.98,155.24,0.00),v40,z0,tPen\WObj:=wPaper;
    MoveL Offs(pOrigin,156.29,138.66,0.00),v40,z0,tPen\WObj:=wPaper;
    MoveL Offs(pOrigin,156.29,137.60,0.00),v40,z0,tPen\WObj:=wPaper;
    MoveL Offs(pOrigin,156.29,137.60,0.00),v40,z0,tPen\WObj:=wPaper;
    MoveL Offs(pOrigin,155.51,137.88,0.00),v40,z0,tPen\WObj:=wPaper;
    MoveL Offs(pOrigin,149.20,145.46,0.00),v40,z0,tPen\WObj:=wPaper;
    MoveL Offs(pOrigin,143.96,150.56,0.00),v40,z0,tPen\WObj:=wPaper;
    MoveL Offs(pOrigin,144.23,150.50,0.00),v40,z0,tPen\WObj:=wPaper;
    MoveL Offs(pOrigin,142.88,149.14,0.00),v40,z0,tPen\WObj:=wPaper;
    MoveL Offs(pOrigin,143.32,149.11,0.00),v40,z0,tPen\WObj:=wPaper;
    MoveL Offs(pOrigin,145.02,149.11,0.00),v40,z0,tPen\WObj:=wPaper;
  ENDPROC

  PROC DrawPart35()
    MoveL Offs(pOrigin,145.24,149.29,0.00),v40,z0,tPen\WObj:=wPaper;
    MoveL Offs(pOrigin,145.66,149.07,0.00),v40,z0,tPen\WObj:=wPaper;
    MoveL Offs(pOrigin,145.24,149.29,0.00),v40,z0,tPen\WObj:=wPaper;
    MoveL Offs(pOrigin,145.13,149.90,0.00),v40,z0,tPen\WObj:=wPaper;
    MoveL Offs(pOrigin,143.62,148.40,0.00),v40,z0,tPen\WObj:=wPaper;
    MoveL Offs(pOrigin,143.54,148.86,0.00),v40,z0,tPen\WObj:=wPaper;
    MoveL Offs(pOrigin,143.32,149.29,0.00),v40,z0,tPen\WObj:=wPaper;
    MoveL Offs(pOrigin,143.54,148.86,0.00),v40,z0,tPen\WObj:=wPaper;
    MoveL Offs(pOrigin,144.18,148.23,0.00),v40,z0,tPen\WObj:=wPaper;
    MoveL Offs(pOrigin,143.96,148.65,0.00),v40,z0,tPen\WObj:=wPaper;
    MoveL Offs(pOrigin,144.18,148.23,0.00),v40,z0,tPen\WObj:=wPaper;
    MoveL Offs(pOrigin,144.60,148.06,0.00),v40,z0,tPen\WObj:=wPaper;
    MoveL Offs(pOrigin,146.30,148.06,0.00),v40,z0,tPen\WObj:=wPaper;
    MoveL Offs(pOrigin,146.30,148.44,0.00),v40,z0,tPen\WObj:=wPaper;
    MoveL Offs(pOrigin,146.51,148.01,0.00),v40,z0,tPen\WObj:=wPaper;
    MoveL Offs(pOrigin,146.30,148.44,0.00),v40,z0,tPen\WObj:=wPaper;
    MoveL Offs(pOrigin,146.62,148.41,0.00),v40,z0,tPen\WObj:=wPaper;
    MoveL Offs(pOrigin,145.12,146.90,0.00),v40,z0,tPen\WObj:=wPaper;
    MoveL Offs(pOrigin,145.45,147.00,0.00),v40,z0,tPen\WObj:=wPaper;
    MoveL Offs(pOrigin,147.36,147.00,0.00),v40,z0,tPen\WObj:=wPaper;
    MoveL Offs(pOrigin,147.79,146.74,0.00),v40,z0,tPen\WObj:=wPaper;
    MoveL Offs(pOrigin,147.57,147.16,0.00),v40,z0,tPen\WObj:=wPaper;
    MoveL Offs(pOrigin,147.79,146.74,0.00),v40,z0,tPen\WObj:=wPaper;
    MoveL Offs(pOrigin,148.26,147.06,0.00),v40,z0,tPen\WObj:=wPaper;
    MoveL Offs(pOrigin,146.61,145.41,0.00),v40,z0,tPen\WObj:=wPaper;
    MoveL Offs(pOrigin,146.73,145.68,0.00),v40,z0,tPen\WObj:=wPaper;
    MoveL Offs(pOrigin,146.51,146.10,0.00),v40,z0,tPen\WObj:=wPaper;
    MoveL Offs(pOrigin,146.73,145.68,0.00),v40,z0,tPen\WObj:=wPaper;
    MoveL Offs(pOrigin,146.51,145.94,0.00),v40,z0,tPen\WObj:=wPaper;
    MoveL Offs(pOrigin,148.43,145.94,0.00),v40,z0,tPen\WObj:=wPaper;
    MoveL Offs(pOrigin,148.43,146.10,0.00),v40,z0,tPen\WObj:=wPaper;
    MoveL Offs(pOrigin,148.21,146.52,0.00),v40,z0,tPen\WObj:=wPaper;
    MoveL Offs(pOrigin,148.43,146.10,0.00),v40,z0,tPen\WObj:=wPaper;
    MoveL Offs(pOrigin,148.86,146.17,0.00),v40,z0,tPen\WObj:=wPaper;
    MoveL Offs(pOrigin,147.36,144.66,0.00),v40,z0,tPen\WObj:=wPaper;
    MoveL Offs(pOrigin,147.57,144.89,0.00),v40,z0,tPen\WObj:=wPaper;
    MoveL Offs(pOrigin,149.28,144.89,0.00),v40,z0,tPen\WObj:=wPaper;
    MoveL Offs(pOrigin,149.49,145.04,0.00),v40,z0,tPen\WObj:=wPaper;
    MoveL Offs(pOrigin,149.70,144.61,0.00),v40,z0,tPen\WObj:=wPaper;
    MoveL Offs(pOrigin,149.49,145.04,0.00),v40,z0,tPen\WObj:=wPaper;
    MoveL Offs(pOrigin,149.76,145.57,0.00),v40,z0,tPen\WObj:=wPaper;
    MoveL Offs(pOrigin,147.95,143.77,0.00),v40,z0,tPen\WObj:=wPaper;
    MoveL Offs(pOrigin,148.43,143.83,0.00),v40,z0,tPen\WObj:=wPaper;
    MoveL Offs(pOrigin,150.34,143.83,0.00),v40,z0,tPen\WObj:=wPaper;
    MoveL Offs(pOrigin,150.76,143.76,0.00),v40,z0,tPen\WObj:=wPaper;
    MoveL Offs(pOrigin,150.98,143.34,0.00),v40,z0,tPen\WObj:=wPaper;
    MoveL Offs(pOrigin,150.76,143.76,0.00),v40,z0,tPen\WObj:=wPaper;
    MoveL Offs(pOrigin,150.95,143.78,0.00),v40,z0,tPen\WObj:=wPaper;
    MoveL Offs(pOrigin,149.45,142.27,0.00),v40,z0,tPen\WObj:=wPaper;
    MoveL Offs(pOrigin,149.49,142.70,0.00),v40,z0,tPen\WObj:=wPaper;
    MoveL Offs(pOrigin,149.27,143.12,0.00),v40,z0,tPen\WObj:=wPaper;
    MoveL Offs(pOrigin,149.49,142.70,0.00),v40,z0,tPen\WObj:=wPaper;
    MoveL Offs(pOrigin,149.49,142.78,0.00),v40,z0,tPen\WObj:=wPaper;
    MoveL Offs(pOrigin,151.19,142.78,0.00),v40,z0,tPen\WObj:=wPaper;
    MoveL Offs(pOrigin,151.61,142.70,0.00),v40,z0,tPen\WObj:=wPaper;
    MoveL Offs(pOrigin,151.82,142.27,0.00),v40,z0,tPen\WObj:=wPaper;
    MoveL Offs(pOrigin,151.61,142.70,0.00),v40,z0,tPen\WObj:=wPaper;
    MoveL Offs(pOrigin,151.70,143.03,0.00),v40,z0,tPen\WObj:=wPaper;
    MoveL Offs(pOrigin,148.54,139.87,0.00),v40,z0,tPen\WObj:=wPaper;
    MoveL Offs(pOrigin,149.44,139.28,0.00),v40,z0,tPen\WObj:=wPaper;
    MoveL Offs(pOrigin,152.44,142.28,0.00),v40,z0,tPen\WObj:=wPaper;
    MoveL Offs(pOrigin,152.25,141.72,0.00),v40,z0,tPen\WObj:=wPaper;
    MoveL Offs(pOrigin,150.34,141.72,0.00),v40,z0,tPen\WObj:=wPaper;
    MoveL Offs(pOrigin,150.34,141.85,0.00),v40,z0,tPen\WObj:=wPaper;
    MoveL Offs(pOrigin,150.55,141.43,0.00),v40,z0,tPen\WObj:=wPaper;
    MoveL Offs(pOrigin,150.34,141.85,0.00),v40,fine,tPen\WObj:=wPaper;
    MoveL Offs(pOrigin,150.34,141.85,6.00),v60,z5,tPen\WObj:=wPaper;
    MoveL Offs(pOrigin,151.19,140.79,6.00),vTravel,z5,tPen\WObj:=wPaper;
    MoveL Offs(pOrigin,151.19,140.79,0.00),v60,z0,tPen\WObj:=wPaper;
    MoveL Offs(pOrigin,150.98,141.21,0.00),v40,z0,tPen\WObj:=wPaper;
    MoveL Offs(pOrigin,151.19,140.79,0.00),v40,z0,tPen\WObj:=wPaper;
    MoveL Offs(pOrigin,151.19,140.66,0.00),v40,z0,tPen\WObj:=wPaper;
    MoveL Offs(pOrigin,153.10,140.66,0.00),v40,z0,tPen\WObj:=wPaper;
    MoveL Offs(pOrigin,153.52,140.36,0.00),v40,z0,tPen\WObj:=wPaper;
    MoveL Offs(pOrigin,153.31,140.79,0.00),v40,z0,tPen\WObj:=wPaper;
    MoveL Offs(pOrigin,153.52,140.36,0.00),v40,z0,tPen\WObj:=wPaper;
    MoveL Offs(pOrigin,153.79,140.64,0.00),v40,z0,tPen\WObj:=wPaper;
    MoveL Offs(pOrigin,151.23,138.08,0.00),v40,z0,tPen\WObj:=wPaper;
    MoveL Offs(pOrigin,151.40,138.45,0.00),v40,z0,tPen\WObj:=wPaper;
    MoveL Offs(pOrigin,151.19,138.66,0.00),v40,z0,tPen\WObj:=wPaper;
    MoveL Offs(pOrigin,151.40,138.24,0.00),v40,z0,tPen\WObj:=wPaper;
    MoveL Offs(pOrigin,152.68,137.81,0.00),v40,z0,tPen\WObj:=wPaper;
    MoveL Offs(pOrigin,152.68,138.02,0.00),v40,z0,tPen\WObj:=wPaper;
    MoveL Offs(pOrigin,152.68,138.02,0.00),v40,z0,tPen\WObj:=wPaper;
    MoveL Offs(pOrigin,152.39,139.51,0.00),v40,z0,tPen\WObj:=wPaper;
    MoveL Offs(pOrigin,148.14,144.40,0.00),v40,z0,tPen\WObj:=wPaper;
    MoveL Offs(pOrigin,142.90,149.64,0.00),v40,z0,tPen\WObj:=wPaper;
    MoveL Offs(pOrigin,138.44,153.11,0.00),v40,z0,tPen\WObj:=wPaper;
    MoveL Offs(pOrigin,137.95,153.17,0.00),v40,z0,tPen\WObj:=wPaper;
    MoveL Offs(pOrigin,139.00,154.22,0.00),v40,z0,tPen\WObj:=wPaper;
    MoveL Offs(pOrigin,139.89,153.63,0.00),v40,z0,tPen\WObj:=wPaper;
    MoveL Offs(pOrigin,138.84,152.58,0.00),v40,z0,tPen\WObj:=wPaper;
    MoveL Offs(pOrigin,137.93,152.04,0.00),v40,z0,tPen\WObj:=wPaper;
    MoveL Offs(pOrigin,135.08,154.89,0.00),v40,z0,tPen\WObj:=wPaper;
    MoveL Offs(pOrigin,134.61,155.02,0.00),v40,z0,tPen\WObj:=wPaper;
    MoveL Offs(pOrigin,137.16,154.39,0.00),v40,z0,tPen\WObj:=wPaper;
    MoveL Offs(pOrigin,137.16,154.39,0.00),v40,z0,tPen\WObj:=wPaper;
    MoveL Offs(pOrigin,138.01,154.39,0.00),v40,z0,tPen\WObj:=wPaper;
    MoveL Offs(pOrigin,139.29,153.82,0.00),v40,z0,tPen\WObj:=wPaper;
    MoveL Offs(pOrigin,143.40,150.85,0.00),v40,z0,tPen\WObj:=wPaper;
    MoveL Offs(pOrigin,142.69,151.41,0.00),v40,z0,tPen\WObj:=wPaper;
    MoveL Offs(pOrigin,142.48,151.22,0.00),v40,z0,tPen\WObj:=wPaper;
    MoveL Offs(pOrigin,141.20,151.22,0.00),v40,z0,tPen\WObj:=wPaper;
    MoveL Offs(pOrigin,140.77,151.41,0.00),v40,z0,tPen\WObj:=wPaper;
    MoveL Offs(pOrigin,141.20,151.20,0.00),v40,z0,tPen\WObj:=wPaper;
    MoveL Offs(pOrigin,140.77,151.41,0.00),v40,z0,tPen\WObj:=wPaper;
    MoveL Offs(pOrigin,140.49,151.23,0.00),v40,z0,tPen\WObj:=wPaper;
    MoveL Offs(pOrigin,141.69,152.44,0.00),v40,z0,tPen\WObj:=wPaper;
    MoveL Offs(pOrigin,140.79,153.03,0.00),v40,z0,tPen\WObj:=wPaper;
    MoveL Offs(pOrigin,139.74,151.98,0.00),v40,z0,tPen\WObj:=wPaper;
    MoveL Offs(pOrigin,140.14,152.05,0.00),v40,z0,tPen\WObj:=wPaper;
    MoveL Offs(pOrigin,140.35,151.62,0.00),v40,z0,tPen\WObj:=wPaper;
    MoveL Offs(pOrigin,140.14,152.05,0.00),v40,fine,tPen\WObj:=wPaper;
    MoveL Offs(pOrigin,140.14,152.05,6.00),v60,z5,tPen\WObj:=wPaper;
    MoveL Offs(pOrigin,141.07,153.38,6.00),vTravel,z5,tPen\WObj:=wPaper;
    MoveL Offs(pOrigin,141.07,153.38,0.00),v60,z0,tPen\WObj:=wPaper;
    MoveL Offs(pOrigin,159.41,135.04,0.00),v40,z0,tPen\WObj:=wPaper;
    MoveL Offs(pOrigin,159.01,135.41,0.00),v40,z0,tPen\WObj:=wPaper;
    MoveL Offs(pOrigin,156.46,132.86,0.00),v40,z0,tPen\WObj:=wPaper;
    MoveL Offs(pOrigin,156.50,133.27,0.00),v40,z0,tPen\WObj:=wPaper;
  ENDPROC

